C01820=1061.236,135.511,-79.537,172.179,30.450,155.636
C01821=1061.242,135.759,-79.557,172.181,30.453,155.636
C01822=1061.248,136.008,-79.578,172.183,30.455,155.637
C01823=1061.253,136.258,-79.599,172.185,30.458,155.637
C01824=1061.259,136.507,-79.619,172.186,30.461,155.638
C01825=1061.266,136.756,-79.641,172.188,30.463,155.638
C01826=1061.271,137.005,-79.661,172.190,30.466,155.638
C01827=1061.278,137.254,-79.682,172.192,30.469,155.639
C01828=1061.283,137.503,-79.703,172.193,30.471,155.639
C01829=1061.289,137.751,-79.724,172.195,30.474,155.640
C01830=1061.295,138.001,-79.745,172.197,30.477,155.640
C01831=1061.300,138.250,-79.765,172.199,30.480,155.640
C01832=1061.307,138.499,-79.787,172.201,30.482,155.641
C01833=1061.313,138.748,-79.807,172.202,30.485,155.641
C01834=1061.319,138.997,-79.828,172.204,30.488,155.642
C01835=1061.324,139.246,-79.849,172.205,30.490,155.642
C01836=1061.331,139.495,-79.870,172.207,30.493,155.643
C01837=1061.336,139.744,-79.891,172.208,30.495,155.643
C01838=1061.342,139.993,-79.912,172.210,30.498,155.643
C01839=1061.348,140.243,-79.933,172.212,30.501,155.644
C01840=1061.353,140.491,-79.954,172.214,30.503,155.644
C01841=1061.360,140.741,-79.974,172.215,30.507,155.645
C01842=1061.365,140.989,-79.996,172.217,30.509,155.645
C01843=1061.371,141.239,-80.017,172.219,30.512,155.646
C01844=1061.377,141.488,-80.038,172.221,30.515,155.646
C01845=1061.383,141.737,-80.059,172.223,30.517,155.646
C01846=1061.388,141.986,-80.080,172.224,30.520,155.647
C01847=1061.395,142.270,-80.104,172.226,30.523,155.647
C01848=1061.402,142.554,-80.128,172.229,30.526,155.648
C01849=1061.409,142.839,-80.152,172.231,30.529,155.648
C01850=1061.416,143.123,-80.176,172.232,30.533,155.649
C01851=1061.421,143.372,-80.197,172.234,30.535,155.649
C01852=1061.427,143.621,-80.219,172.236,30.538,155.650
C01853=1061.433,143.870,-80.240,172.238,30.541,155.650
C01854=1061.438,144.120,-80.261,172.239,30.543,155.650
C01855=1061.444,144.368,-80.282,172.241,30.546,155.651
C01856=1061.450,144.617,-80.304,172.243,30.549,155.651
C01857=1061.455,144.866,-80.324,172.245,30.551,155.652
C01858=1061.462,145.115,-80.345,172.246,30.554,155.652
C01859=1061.468,145.364,-80.367,172.248,30.557,155.653
C01860=1061.474,145.613,-80.388,172.250,30.560,155.653
C01861=1061.480,145.863,-80.409,172.252,30.563,155.653
C01862=1061.486,146.111,-80.430,172.254,30.565,155.654
C01863=1061.492,146.361,-80.452,172.255,30.568,155.654
C01864=1061.497,146.610,-80.473,172.257,30.571,155.655
C01865=1061.503,146.859,-80.494,172.259,30.573,155.655
C01866=1061.509,147.107,-80.515,172.261,30.576,155.655
C01867=1061.515,147.357,-80.537,172.262,30.579,155.656
C01868=1061.522,147.605,-80.558,172.264,30.581,155.656
C01869=1061.527,147.855,-80.579,172.266,30.584,155.657
C01870=1061.532,148.104,-80.601,172.268,30.587,155.657
C01871=1061.538,148.353,-80.622,172.270,30.590,155.658
C01872=1061.544,148.602,-80.644,172.271,30.592,155.658
C01873=1061.550,148.850,-80.665,172.273,30.595,155.658
C01874=1061.556,149.100,-80.687,172.275,30.598,155.659
C01875=1061.562,149.349,-80.708,172.277,30.600,155.659
C01876=1061.567,149.598,-80.729,172.278,30.603,155.660
C01877=1061.573,149.847,-80.751,172.280,30.606,155.660
C01878=1061.579,150.096,-80.772,172.282,30.609,155.661
C01879=1061.585,150.345,-80.793,172.284,30.612,155.661
C01880=1061.591,150.594,-80.815,172.286,30.614,155.662
C01881=1061.597,150.843,-80.836,172.287,30.617,155.662
C01882=1061.603,151.092,-80.858,172.289,30.620,155.662
C01883=1061.608,151.341,-80.880,172.291,30.622,155.663
C01884=1061.614,151.590,-80.901,172.294,30.625,155.663
C01885=1061.620,151.839,-80.923,172.295,30.628,155.664
C01886=1061.626,152.087,-80.944,172.297,30.631,155.664
C01887=1061.632,152.337,-80.966,172.299,30.634,155.665
C01888=1061.637,152.585,-80.987,172.301,30.636,155.665
C01889=1061.644,152.834,-81.009,172.302,30.639,155.665
C01890=1061.649,153.084,-81.031,172.304,30.642,155.666
C01891=1061.655,153.332,-81.052,172.306,30.645,155.666
C01892=1061.661,153.582,-81.074,172.308,30.648,155.667
C01893=1061.667,153.831,-81.096,172.310,30.650,155.667
C01894=1061.673,154.079,-81.117,172.311,30.653,155.668
C01895=1061.679,154.329,-81.139,172.313,30.656,155.668
C01896=1061.684,154.578,-81.161,172.315,30.658,155.668
C01897=1061.690,154.827,-81.182,172.317,30.661,155.669
C01898=1061.696,155.076,-81.204,172.318,30.664,155.669
C01899=1061.702,155.325,-81.225,172.320,30.667,155.670
C01900=1061.708,155.573,-81.247,172.322,30.669,155.670
C01901=1061.713,155.822,-81.270,172.324,30.672,155.671
C01902=1061.719,156.072,-81.291,172.326,30.675,155.671
C01903=1061.726,156.321,-81.313,172.327,30.678,155.671
C01904=1061.730,156.570,-81.335,172.330,30.681,155.672
C01905=1061.737,156.819,-81.356,172.332,30.684,155.672
C01906=1061.743,157.068,-81.378,172.334,30.686,155.673
C01907=1061.748,157.316,-81.401,172.336,30.689,155.673
C01908=1061.754,157.565,-81.422,172.337,30.692,155.674
C01909=1061.760,157.815,-81.444,172.339,30.695,155.674
C01910=1061.766,158.063,-81.465,172.341,30.697,155.675
C01911=1061.773,158.348,-81.491,172.343,30.701,155.675
C01912=1061.779,158.631,-81.516,172.345,30.704,155.676
C01913=1061.786,158.915,-81.540,172.347,30.707,155.676
C01914=1061.793,159.200,-81.566,172.349,30.710,155.676
C01915=1061.798,159.448,-81.587,172.351,30.713,155.677
C01916=1061.804,159.698,-81.609,172.353,30.716,155.677
C01917=1061.810,159.946,-81.632,172.355,30.719,155.678
C01918=1061.816,160.196,-81.653,172.357,30.721,155.678
C01919=1061.821,160.444,-81.675,172.359,30.724,155.679
C01920=1061.827,160.693,-81.697,172.361,30.727,155.679
C01921=1061.834,160.942,-81.719,172.362,30.729,155.679
C01922=1061.839,161.192,-81.741,172.364,30.732,155.680
C01923=1061.845,161.440,-81.763,172.366,30.735,155.680
C01924=1061.850,161.689,-81.786,172.368,30.738,155.681
C01925=1061.856,161.938,-81.809,172.369,30.741,155.681
C01926=1061.862,162.187,-81.830,172.371,30.744,155.682
C01927=1061.867,162.436,-81.852,172.374,30.747,155.682
C01928=1061.873,162.685,-81.875,172.376,30.750,155.683
C01929=1061.879,162.934,-81.897,172.378,30.752,155.683
C01930=1061.884,163.182,-81.919,172.379,30.756,155.684
C01931=1061.889,163.432,-81.941,172.381,30.758,155.684
C01932=1061.896,163.680,-81.964,172.383,30.761,155.685
C01933=1061.901,163.930,-81.986,172.385,30.764,155.685
C01934=1061.907,164.178,-82.009,172.386,30.767,155.685
C01935=1061.913,164.427,-82.030,172.388,30.770,155.686
C01936=1061.918,164.676,-82.053,172.390,30.773,155.686
C01937=1061.924,164.926,-82.075,172.393,30.775,155.687
C01938=1061.929,165.174,-82.098,172.395,30.779,155.687
C01939=1061.935,165.423,-82.120,172.396,30.781,155.688
C01940=1061.941,165.672,-82.143,172.398,30.785,155.688
C01941=1061.946,165.922,-82.165,172.400,30.787,155.689
C01942=1061.952,166.169,-82.187,172.402,30.790,155.689
C01943=1061.958,166.419,-82.209,172.403,30.793,155.690
C01944=1061.963,166.668,-82.232,172.405,30.796,155.690
C01945=1061.970,166.916,-82.254,172.407,30.798,155.691
C01946=1061.975,167.166,-82.277,172.410,30.802,155.691
C01947=1061.981,167.415,-82.299,172.412,30.804,155.691
C01948=1061.986,167.664,-82.321,172.413,30.808,155.692
C01949=1061.992,167.912,-82.344,172.415,30.810,155.692
C01950=1061.998,168.161,-82.367,172.417,30.813,155.693
C01951=1062.003,168.411,-82.389,172.419,30.816,155.693
C01952=1062.009,168.660,-82.412,172.421,30.819,155.694
C01953=1062.016,168.908,-82.434,172.423,30.822,155.694
C01954=1062.020,169.157,-82.456,172.425,30.825,155.695
C01955=1062.026,169.406,-82.479,172.427,30.827,155.695
C01956=1062.033,169.654,-82.501,172.429,30.830,155.696
C01957=1062.038,169.904,-82.524,172.430,30.833,155.696
C01958=1062.044,170.153,-82.546,172.432,30.836,155.696
C01959=1062.049,170.402,-82.569,172.434,30.839,155.697
C01960=1062.055,170.651,-82.592,172.437,30.842,155.697
C01961=1062.061,170.900,-82.614,172.439,30.845,155.698
C01962=1062.067,171.148,-82.637,172.440,30.848,155.698
C01963=1062.072,171.397,-82.660,172.442,30.850,155.699
C01964=1062.078,171.646,-82.682,172.444,30.853,155.699
C01965=1062.084,171.895,-82.704,172.446,30.856,155.700
C01966=1062.090,172.144,-82.727,172.448,30.859,155.700
C01967=1062.096,172.393,-82.750,172.450,30.862,155.701
C01968=1062.101,172.642,-82.773,172.452,30.865,155.701
C01969=1062.108,172.890,-82.795,172.454,30.868,155.702
C01970=1062.113,173.140,-82.818,172.456,30.871,155.702
C01971=1062.119,173.389,-82.840,172.457,30.874,155.702
C01972=1062.125,173.638,-82.863,172.460,30.876,155.703
C01973=1062.130,173.887,-82.886,172.462,30.880,155.703
C01974=1062.137,174.135,-82.909,172.464,30.882,155.704
C01975=1062.143,174.419,-82.934,172.467,30.886,155.704
C01976=1062.150,174.703,-82.960,172.468,30.889,155.705
C01977=1062.156,174.986,-82.987,172.471,30.892,155.705
C01978=1062.163,175.270,-83.012,172.473,30.895,155.706
C01979=1062.169,175.518,-83.035,172.475,30.898,155.706
C01980=1062.175,175.767,-83.058,172.476,30.901,155.707
C01981=1062.180,176.016,-83.081,172.479,30.904,155.707
C01982=1062.186,176.265,-83.104,172.481,30.907,155.708
C01983=1062.192,176.514,-83.126,172.483,30.910,155.708
C01984=1062.198,176.763,-83.149,172.485,30.912,155.709
C01985=1062.204,177.012,-83.172,172.486,30.915,155.709
C01986=1062.210,177.261,-83.195,172.489,30.919,155.710
C01987=1062.216,177.510,-83.218,172.491,30.921,155.710
C01988=1062.222,177.759,-83.241,172.493,30.924,155.710
C01989=1062.228,178.008,-83.264,172.495,30.927,155.711
C01990=1062.233,178.257,-83.287,172.497,30.930,155.711
C01991=1062.240,178.505,-83.309,172.499,30.932,155.712
C01992=1062.246,178.754,-83.332,172.501,30.936,155.712
C01993=1062.251,179.003,-83.355,172.503,30.938,155.713
C01994=1062.257,179.252,-83.378,172.505,30.941,155.713
C01995=1062.263,179.501,-83.401,172.507,30.944,155.714
C01996=1062.269,179.749,-83.425,172.509,30.947,155.714
C01997=1062.275,179.998,-83.447,172.511,30.950,155.715
C01998=1062.282,180.247,-83.470,172.513,30.953,155.715
C01999=1062.287,180.496,-83.493,172.516,30.956,155.715
C02000=1062.293,180.745,-83.516,172.517,30.959,155.716
C02001=1062.299,180.994,-83.539,172.519,30.961,155.716
C02002=1062.305,181.243,-83.562,172.521,30.964,155.717
C02003=1062.311,181.491,-83.586,172.524,30.967,155.717
C02004=1062.316,181.740,-83.609,172.525,30.970,155.718
C02005=1062.323,181.989,-83.631,172.527,30.973,155.718
C02006=1062.329,182.238,-83.654,172.529,30.976,155.719
C02007=1062.335,182.487,-83.677,172.532,30.979,155.719
C02008=1062.341,182.735,-83.701,172.534,30.981,155.720
C02009=1062.347,182.984,-83.724,172.535,30.984,155.720
C02010=1062.353,183.234,-83.747,172.538,30.987,155.720
C02011=1062.359,183.483,-83.770,172.540,30.990,155.721
C02012=1062.364,183.732,-83.793,172.542,30.993,155.721
C02013=1062.370,183.980,-83.817,172.544,30.996,155.722
C02014=1062.376,184.229,-83.840,172.546,30.999,155.722
C02015=1062.383,184.478,-83.862,172.548,31.002,155.723
C02016=1062.389,184.727,-83.887,172.550,31.005,155.723
C02017=1062.394,184.976,-83.910,172.552,31.008,155.724
C02018=1062.399,185.225,-83.933,172.555,31.011,155.724
C02019=1062.405,185.473,-83.957,172.556,31.014,155.725
C02020=1062.411,185.722,-83.980,172.558,31.017,155.725
C02021=1062.416,185.971,-84.004,172.561,31.020,155.726
C02022=1062.422,186.220,-84.027,172.563,31.023,155.726
C02023=1062.428,186.469,-84.050,172.565,31.026,155.727
C02024=1062.434,186.718,-84.075,172.566,31.029,155.727
C02025=1062.439,186.967,-84.098,172.569,31.032,155.728
C02026=1062.445,187.215,-84.121,172.571,31.035,155.728
C02027=1062.450,187.464,-84.145,172.573,31.038,155.729
C02028=1062.456,187.712,-84.168,172.575,31.041,155.729
C02029=1062.461,187.962,-84.192,172.577,31.044,155.730
C02030=1062.468,188.211,-84.216,172.579,31.048,155.730
C02031=1062.474,188.459,-84.239,172.581,31.050,155.731
C02032=1062.479,188.708,-84.263,172.584,31.053,155.731
C02033=1062.485,188.957,-84.286,172.585,31.057,155.732
C02034=1062.490,189.206,-84.310,172.587,31.059,155.732
C02035=1062.496,189.454,-84.333,172.590,31.063,155.733
C02036=1062.503,189.703,-84.357,172.592,31.066,155.733
C02037=1062.508,189.952,-84.382,172.594,31.068,155.734
C02038=1062.514,190.201,-84.405,172.595,31.072,155.734
C02039=1062.520,190.484,-84.432,172.598,31.075,155.735
C02040=1062.527,190.768,-84.458,172.601,31.079,155.735
C02041=1062.533,191.050,-84.486,172.603,31.082,155.736
C02042=1062.540,191.334,-84.513,172.606,31.086,155.736
C02043=1062.546,191.583,-84.536,172.607,31.089,155.737
C02044=1062.551,191.831,-84.561,172.610,31.091,155.737
C02045=1062.557,192.080,-84.584,172.612,31.095,155.738
C02046=1062.563,192.329,-84.608,172.614,31.098,155.738
C02047=1062.569,192.578,-84.632,172.617,31.101,155.739
C02048=1062.575,192.826,-84.655,172.618,31.104,155.739
C02049=1062.580,193.075,-84.679,172.620,31.107,155.740
C02050=1062.586,193.324,-84.703,172.623,31.110,155.740
C02051=1062.591,193.573,-84.727,172.625,31.113,155.741
C02052=1062.597,193.822,-84.750,172.627,31.116,155.741
C02053=1062.603,194.071,-84.775,172.629,31.120,155.742
C02054=1062.609,194.319,-84.798,172.631,31.122,155.742
C02055=1062.615,194.568,-84.822,172.633,31.125,155.743
C02056=1062.621,194.817,-84.847,172.636,31.129,155.743
C02057=1062.627,195.066,-84.870,172.638,31.131,155.744
C02058=1062.632,195.314,-84.894,172.639,31.135,155.744
C02059=1062.639,195.563,-84.918,172.642,31.138,155.745
C02060=1062.644,195.812,-84.942,172.644,31.140,155.745
C02061=1062.650,196.060,-84.966,172.647,31.144,155.746
C02062=1062.656,196.310,-84.990,172.649,31.147,155.746
C02063=1062.662,196.558,-85.013,172.650,31.150,155.747
C02064=1062.668,196.808,-85.038,172.653,31.153,155.747
C02065=1062.674,197.056,-85.062,172.655,31.156,155.748
C02066=1062.679,197.305,-85.086,172.657,31.159,155.748
C02067=1062.686,197.554,-85.110,172.660,31.162,155.749
C02068=1062.691,197.802,-85.134,172.661,31.165,155.749
C02069=1062.697,198.050,-85.158,172.664,31.169,155.750
C02070=1062.703,198.300,-85.183,172.666,31.171,155.750
C02071=1062.709,198.548,-85.206,172.668,31.174,155.751
C02072=1062.714,198.798,-85.230,172.671,31.178,155.751
C02073=1062.720,199.046,-85.254,172.672,31.180,155.752
C02074=1062.726,199.295,-85.278,172.675,31.184,155.752
C02075=1062.732,199.544,-85.302,172.677,31.187,155.753
C02076=1062.738,199.793,-85.327,172.679,31.190,155.753
C02077=1062.744,200.041,-85.350,172.682,31.193,155.754
C02078=1062.750,200.290,-85.375,172.683,31.196,155.754
C02079=1062.756,200.539,-85.399,172.686,31.199,155.755
C02080=1062.762,200.787,-85.424,172.688,31.202,155.755
C02081=1062.768,201.036,-85.448,172.690,31.205,155.756
C02082=1062.774,201.284,-85.472,172.693,31.209,155.756
C02083=1062.780,201.534,-85.497,172.694,31.211,155.757
C02084=1062.786,201.782,-85.520,172.697,31.214,155.757
C02085=1062.792,202.031,-85.545,172.699,31.218,155.758
C02086=1062.797,202.280,-85.569,172.702,31.221,155.758
C02087=1062.804,202.529,-85.593,172.704,31.224,155.759
C02088=1062.809,202.777,-85.617,172.705,31.227,155.759
C02089=1062.815,203.026,-85.643,172.708,31.230,155.760
C02090=1062.820,203.275,-85.667,172.710,31.233,155.760
C02091=1062.826,203.524,-85.692,172.713,31.237,155.761
C02092=1062.832,203.772,-85.715,172.715,31.240,155.761
C02093=1062.838,204.021,-85.740,172.717,31.243,155.762
C02094=1062.844,204.269,-85.765,172.719,31.246,155.763
C02095=1062.850,204.519,-85.789,172.721,31.250,155.763
C02096=1062.855,204.767,-85.814,172.724,31.253,155.764
C02097=1062.861,205.017,-85.838,172.726,31.256,155.764
C02098=1062.867,205.264,-85.863,172.728,31.259,155.765
C02099=1062.873,205.514,-85.887,172.730,31.262,155.765
C02100=1062.879,205.762,-85.912,172.733,31.265,155.766
C02101=1062.884,206.011,-85.936,172.735,31.268,155.766
C02102=1062.890,206.259,-85.961,172.738,31.272,155.767
C02103=1062.915,207.308,-86.065,172.906,31.353,155.774
C02104=1062.920,207.532,-86.088,172.908,31.357,155.775
C02105=1062.926,207.757,-86.110,172.910,31.361,155.775
C02106=1062.931,207.982,-86.134,172.911,31.364,155.776
C02107=1062.937,208.207,-86.156,172.913,31.368,155.777
C02108=1062.943,208.432,-86.179,172.915,31.372,155.777
C02109=1062.948,208.657,-86.203,172.917,31.376,155.778
C02110=1062.953,208.881,-86.225,172.919,31.379,155.779
C02111=1062.959,209.107,-86.248,172.920,31.383,155.779
C02112=1062.965,209.355,-86.274,172.922,31.387,155.780
C02113=1062.971,209.604,-86.300,172.924,31.391,155.781
C02114=1062.977,209.852,-86.326,172.926,31.395,155.782
C02115=1062.983,210.101,-86.351,172.928,31.399,155.782
C02116=1062.989,210.350,-86.376,172.930,31.404,155.783
C02117=1062.996,210.598,-86.402,172.932,31.407,155.784
C02118=1063.001,210.847,-86.428,172.934,31.412,155.784
C02119=1063.008,211.095,-86.454,172.936,31.415,155.785
C02120=1063.014,211.344,-86.479,172.937,31.420,155.786
C02121=1063.019,211.593,-86.505,172.939,31.423,155.787
C02122=1063.025,211.842,-86.530,172.942,31.428,155.787
C02123=1063.032,212.090,-86.556,172.944,31.432,155.788
C02124=1063.038,212.338,-86.582,172.946,31.436,155.789
C02125=1063.044,212.587,-86.608,172.947,31.440,155.790
C02126=1063.050,212.836,-86.633,172.949,31.444,155.790
C02127=1063.055,213.085,-86.659,172.952,31.448,155.791
C02128=1063.062,213.333,-86.685,172.954,31.452,155.792
C02129=1063.068,213.582,-86.710,172.956,31.456,155.792
C02130=1063.073,213.831,-86.736,172.957,31.460,155.793
C02131=1063.080,214.079,-86.762,172.959,31.464,155.794
C02132=1063.085,214.328,-86.788,172.962,31.469,155.795
C02133=1063.092,214.576,-86.814,172.964,31.472,155.795
C02134=1063.097,214.825,-86.840,172.966,31.477,155.796
C02135=1063.104,215.073,-86.866,172.967,31.480,155.797
C02136=1063.109,215.322,-86.892,172.969,31.485,155.798
C02137=1063.116,215.570,-86.918,172.972,31.488,155.798
C02138=1063.122,215.819,-86.943,172.974,31.493,155.799
C02139=1063.128,216.068,-86.969,172.976,31.496,155.800
C02140=1063.134,216.316,-86.995,172.977,31.501,155.801
C02141=1063.140,216.565,-87.021,172.979,31.504,155.801
C02142=1063.146,216.813,-87.047,172.982,31.509,155.802
C02143=1063.152,217.062,-87.073,172.984,31.513,155.803
C02144=1063.158,217.310,-87.099,172.986,31.517,155.803
C02145=1063.164,217.559,-87.125,172.987,31.521,155.804
C02146=1063.170,217.808,-87.151,172.990,31.525,155.805
C02147=1063.176,218.056,-87.178,172.992,31.529,155.806
C02148=1063.182,218.305,-87.203,172.994,31.533,155.806
C02149=1063.188,218.553,-87.230,172.996,31.537,155.807
C02150=1063.194,218.802,-87.255,172.998,31.541,155.808
C02151=1063.200,219.050,-87.282,173.000,31.545,155.808
C02152=1063.206,219.299,-87.307,173.002,31.549,155.809
C02153=1063.212,219.547,-87.334,173.004,31.553,155.810
C02154=1063.219,219.797,-87.359,173.007,31.557,155.811
C02155=1063.225,220.045,-87.386,173.008,31.561,155.811
C02156=1063.231,220.293,-87.412,173.010,31.565,155.812
C02157=1063.237,220.542,-87.438,173.012,31.569,155.813
C02158=1063.243,220.790,-87.464,173.015,31.573,155.813
C02159=1063.249,221.039,-87.491,173.017,31.577,155.814
C02160=1063.254,221.266,-87.515,173.019,31.581,155.815
C02161=1063.260,221.494,-87.539,173.020,31.584,155.815
C02162=1063.265,221.721,-87.562,173.022,31.588,155.816
C02163=1063.271,221.948,-87.587,173.024,31.591,155.817
C02164=1063.277,222.176,-87.611,173.026,31.595,155.817
C02165=1063.282,222.403,-87.635,173.028,31.599,155.818
C02166=1063.288,222.630,-87.659,173.030,31.602,155.819
C02167=1063.293,222.858,-87.683,173.031,31.606,155.820
C02168=1063.299,223.106,-87.710,173.034,31.611,155.820
C02169=1063.305,223.355,-87.736,173.036,31.614,155.821
C02170=1063.310,223.603,-87.763,173.038,31.619,155.822
C02171=1063.318,223.852,-87.789,173.041,31.622,155.822
C02172=1063.323,224.100,-87.816,173.042,31.627,155.823
C02173=1063.329,224.349,-87.842,173.044,31.630,155.824
C02174=1063.335,224.598,-87.868,173.046,31.635,155.825
C02175=1063.341,224.846,-87.894,173.049,31.638,155.825
C02176=1063.347,225.095,-87.921,173.051,31.642,155.826
C02177=1063.353,225.343,-87.948,173.053,31.646,155.827
C02178=1063.359,225.592,-87.975,173.055,31.650,155.827
C02179=1063.365,225.840,-88.001,173.057,31.655,155.828
C02180=1063.372,226.089,-88.028,173.059,31.658,155.829
C02181=1063.378,226.337,-88.054,173.061,31.662,155.830
C02182=1063.383,226.585,-88.081,173.064,31.666,155.830
C02183=1063.389,226.834,-88.108,173.066,31.670,155.831
C02184=1063.395,227.084,-88.134,173.067,31.674,155.832
C02185=1063.402,227.332,-88.160,173.070,31.678,155.832
C02186=1063.408,227.580,-88.187,173.072,31.682,155.833
C02187=1063.414,227.829,-88.214,173.074,31.686,155.834
C02188=1063.420,228.077,-88.240,173.077,31.690,155.835
C02189=1063.425,228.326,-88.267,173.078,31.694,155.835
C02190=1063.433,228.574,-88.293,173.080,31.698,155.836
C02191=1063.439,228.822,-88.321,173.083,31.702,155.837
C02192=1063.444,229.071,-88.347,173.085,31.706,155.838
C02193=1063.451,229.320,-88.374,173.087,31.710,155.838
C02194=1063.457,229.568,-88.401,173.090,31.714,155.839
C02195=1063.462,229.816,-88.428,173.091,31.718,155.840
C02196=1063.469,230.065,-88.455,173.093,31.721,155.840
C02197=1063.475,230.314,-88.481,173.096,31.726,155.841
C02198=1063.480,230.562,-88.508,173.098,31.730,155.842
C02199=1063.487,230.811,-88.535,173.100,31.734,155.843
C02200=1063.492,231.060,-88.562,173.103,31.738,155.843
C02201=1063.499,231.307,-88.589,173.104,31.742,155.844
C02202=1063.505,231.556,-88.616,173.106,31.746,155.845
C02203=1063.511,231.805,-88.643,173.109,31.749,155.845
C02204=1063.516,232.053,-88.669,173.111,31.754,155.846
C02205=1063.523,232.302,-88.696,173.113,31.757,155.847
C02206=1063.529,232.550,-88.724,173.116,31.762,155.848
C02207=1063.535,232.798,-88.750,173.117,31.765,155.848
C02208=1063.541,233.047,-88.777,173.119,31.770,155.849
C02209=1063.547,233.296,-88.804,173.122,31.774,155.850
C02210=1063.553,233.544,-88.832,173.124,31.777,155.850
C02211=1063.559,233.792,-88.858,173.127,31.782,155.851
C02212=1063.564,234.041,-88.886,173.129,31.785,155.852
C02213=1063.571,234.290,-88.913,173.131,31.790,155.853
C02214=1063.577,234.538,-88.940,173.133,31.793,155.853
C02215=1063.583,234.786,-88.967,173.135,31.798,155.854
C02216=1063.588,235.010,-88.991,173.137,31.801,155.855
C02217=1063.594,235.233,-89.016,173.139,31.804,155.855
C02218=1063.599,235.457,-89.040,173.141,31.808,155.856
C02219=1063.605,235.680,-89.064,173.144,31.812,155.857
C02220=1063.610,235.903,-89.089,173.146,31.815,155.857
C02221=1063.616,236.127,-89.113,173.147,31.819,155.858
C02222=1063.621,236.350,-89.138,173.149,31.822,155.859
C02223=1063.626,236.574,-89.163,173.151,31.826,155.859
C02224=1063.632,236.821,-89.190,173.154,31.830,155.860
C02225=1063.638,237.070,-89.217,173.156,31.834,155.861
C02226=1063.644,237.318,-89.244,173.158,31.838,155.861
C02227=1063.651,237.567,-89.271,173.160,31.842,155.862
C02228=1063.657,237.815,-89.299,173.162,31.846,155.863
C02229=1063.662,238.064,-89.326,173.165,31.850,155.864
C02230=1063.669,238.312,-89.354,173.167,31.853,155.864
C02231=1063.675,238.561,-89.381,173.169,31.858,155.865
C02232=1063.681,238.809,-89.408,173.172,31.861,155.866
C02233=1063.687,239.058,-89.437,173.174,31.865,155.866
C02234=1063.693,239.306,-89.463,173.176,31.869,155.867
C02235=1063.699,239.554,-89.491,173.178,31.873,155.868
C02236=1063.705,239.803,-89.518,173.180,31.877,155.868
C02237=1063.711,240.052,-89.546,173.183,31.881,155.869
C02238=1063.717,240.299,-89.573,173.185,31.885,155.870
C02239=1063.724,240.548,-89.600,173.188,31.889,155.871
C02240=1063.729,240.796,-89.628,173.190,31.893,155.871
C02241=1063.736,241.045,-89.656,173.192,31.897,155.872
C02242=1063.742,241.294,-89.683,173.194,31.900,155.873
C02243=1063.748,241.542,-89.710,173.197,31.905,155.874
C02244=1063.754,241.790,-89.739,173.199,31.908,155.874
C02245=1063.760,242.039,-89.765,173.201,31.912,155.875
C02246=1063.766,242.287,-89.793,173.204,31.917,155.876
C02247=1063.772,242.535,-89.821,173.206,31.920,155.876
C02248=1063.778,242.784,-89.849,173.208,31.925,155.877
C02249=1063.784,243.033,-89.876,173.210,31.928,155.878
C02250=1063.790,243.281,-89.904,173.213,31.932,155.878
C02251=1063.796,243.530,-89.932,173.215,31.936,155.879
C02252=1063.802,243.777,-89.959,173.218,31.940,155.880
C02253=1063.808,244.026,-89.988,173.220,31.944,155.881
C02254=1063.814,244.274,-90.014,173.222,31.948,155.881
C02255=1063.820,244.523,-90.043,173.224,31.952,155.882
C02256=1063.827,244.772,-90.070,173.226,31.956,155.883
C02257=1063.832,245.020,-90.098,173.229,31.960,155.884
C02258=1063.839,245.268,-90.126,173.231,31.964,155.884
C02259=1063.844,245.516,-90.154,173.234,31.968,155.885
C02260=1063.851,245.765,-90.182,173.236,31.972,155.886
C02261=1063.857,246.013,-90.210,173.239,31.976,155.886
C02262=1063.862,246.261,-90.238,173.241,31.980,155.887
C02263=1063.869,246.510,-90.266,173.243,31.984,155.888
C02264=1063.874,246.758,-90.294,173.245,31.988,155.889
C02265=1063.880,247.007,-90.322,173.248,31.992,155.889
C02266=1063.886,247.255,-90.350,173.250,31.996,155.890
C02267=1063.892,247.503,-90.378,173.253,32.000,155.891
C02268=1063.898,247.752,-90.406,173.255,32.004,155.892
C02269=1063.904,248.000,-90.433,173.257,32.007,155.892
C02270=1063.910,248.248,-90.462,173.259,32.012,155.893
C02271=1063.916,248.497,-90.490,173.261,32.015,155.894
C02272=1063.921,248.717,-90.515,173.264,32.019,155.894
C02273=1063.926,248.937,-90.540,173.266,32.023,155.895
C02274=1063.932,249.157,-90.565,173.268,32.026,155.896
C02275=1063.937,249.378,-90.590,173.270,32.030,155.896
C02276=1063.942,249.598,-90.614,173.272,32.033,155.897
C02277=1063.947,249.818,-90.640,173.275,32.037,155.898
C02278=1063.953,250.038,-90.664,173.277,32.040,155.898
C02279=1063.957,250.259,-90.689,173.278,32.044,155.899
C02280=1063.964,250.507,-90.718,173.281,32.048,155.900
C02281=1063.970,250.755,-90.746,173.283,32.052,155.900
C02282=1063.976,251.003,-90.774,173.286,32.056,155.901
C02283=1063.982,251.252,-90.802,173.288,32.060,155.902
C02284=1063.988,251.500,-90.832,173.291,32.064,155.902
C02285=1063.993,251.748,-90.859,173.293,32.068,155.903
C02286=1064.000,251.997,-90.887,173.296,32.072,155.904
C02287=1064.006,252.246,-90.916,173.297,32.076,155.905
C02288=1064.012,252.493,-90.944,173.300,32.080,155.905
C02289=1064.017,252.742,-90.973,173.302,32.083,155.906
C02290=1064.023,252.991,-91.001,173.305,32.088,155.907
C02291=1064.030,253.238,-91.029,173.307,32.091,155.908
C02292=1064.036,253.487,-91.058,173.310,32.096,155.908
C02293=1064.042,253.735,-91.086,173.312,32.099,155.909
C02294=1064.048,253.983,-91.115,173.315,32.103,155.910
C02295=1064.054,254.232,-91.143,173.317,32.107,155.911
C02296=1064.060,254.481,-91.171,173.319,32.111,155.911
C02297=1064.066,254.728,-91.199,173.322,32.115,155.912
C02298=1064.072,254.977,-91.228,173.324,32.119,155.913
C02299=1064.078,255.225,-91.257,173.327,32.123,155.913
C02300=1064.084,255.474,-91.285,173.329,32.127,155.914
C02301=1064.091,255.722,-91.314,173.332,32.131,155.915
C02302=1064.097,255.970,-91.342,173.335,32.135,155.915
C02303=1064.102,256.218,-91.371,173.337,32.139,155.916
C02304=1064.109,256.466,-91.399,173.339,32.143,155.917
C02305=1064.115,256.714,-91.428,173.341,32.146,155.918
C02306=1064.121,256.963,-91.456,173.344,32.151,155.918
C02307=1064.127,257.211,-91.485,173.346,32.154,155.919
C02308=1064.133,257.460,-91.514,173.349,32.158,155.920
C02309=1064.140,257.708,-91.543,173.352,32.162,155.921
C02310=1064.145,257.957,-91.571,173.354,32.166,155.921
C02311=1064.151,258.204,-91.600,173.357,32.170,155.922
C02312=1064.158,258.453,-91.627,173.359,32.174,155.923
C02313=1064.164,258.701,-91.656,173.361,32.178,155.923
C02314=1064.170,258.949,-91.685,173.364,32.181,155.924
C02315=1064.176,259.198,-91.714,173.366,32.186,155.925
C02316=1064.182,259.446,-91.743,173.369,32.189,155.926
C02317=1064.189,259.694,-91.772,173.371,32.193,155.926
C02318=1064.195,259.943,-91.800,173.374,32.197,155.927
C02319=1064.201,260.191,-91.829,173.377,32.201,155.928
C02320=1064.207,260.439,-91.858,173.379,32.205,155.928
C02321=1064.213,260.688,-91.887,173.382,32.209,155.929
C02322=1064.220,260.936,-91.915,173.384,32.213,155.930
C02323=1064.226,261.184,-91.944,173.386,32.217,155.931
C02324=1064.233,261.432,-91.973,173.389,32.220,155.931
C02325=1064.239,261.681,-92.001,173.391,32.225,155.932
C02326=1064.245,261.929,-92.030,173.394,32.228,155.933
C02327=1064.251,262.177,-92.059,173.397,32.232,155.933
C02328=1064.257,262.397,-92.085,173.399,32.236,155.934
C02329=1064.262,262.615,-92.111,173.401,32.239,155.935
C02330=1064.267,262.835,-92.136,173.404,32.243,155.935
C02331=1064.273,263.053,-92.161,173.406,32.246,155.936
C02332=1064.278,263.273,-92.187,173.408,32.249,155.937
C02333=1064.284,263.492,-92.213,173.410,32.252,155.937
C02334=1064.289,263.711,-92.238,173.412,32.256,155.938
C02335=1064.295,263.930,-92.264,173.414,32.260,155.938
C02336=1064.301,264.178,-92.293,173.417,32.263,155.939
C02337=1064.307,264.426,-92.322,173.420,32.268,155.940
C02338=1064.313,264.675,-92.352,173.422,32.271,155.941
C02339=1064.319,264.923,-92.381,173.425,32.276,155.941
C02340=1064.325,265.171,-92.410,173.428,32.280,155.942
C02341=1064.332,265.419,-92.439,173.430,32.283,155.943
C02342=1064.337,265.668,-92.469,173.433,32.287,155.944
C02343=1064.343,265.916,-92.498,173.436,32.291,155.944
C02344=1064.350,266.164,-92.527,173.437,32.295,155.945
C02345=1064.356,266.412,-92.556,173.440,32.299,155.946
C02346=1064.361,266.660,-92.586,173.443,32.303,155.946
C02347=1064.368,266.908,-92.615,173.445,32.307,155.947
C02348=1064.374,267.157,-92.644,173.448,32.311,155.948
C02349=1064.379,267.405,-92.673,173.451,32.315,155.949
C02350=1064.386,267.653,-92.702,173.453,32.319,155.949
C02351=1064.392,267.901,-92.731,173.456,32.323,155.950
C02352=1064.398,268.149,-92.762,173.459,32.327,155.951
C02353=1064.404,268.397,-92.791,173.461,32.331,155.952
C02354=1064.410,268.645,-92.820,173.464,32.335,155.952
C02355=1064.417,268.894,-92.849,173.466,32.339,155.953
C02356=1064.422,269.143,-92.879,173.468,32.343,155.954
C02357=1064.429,269.391,-92.908,173.471,32.347,155.954
C02358=1064.435,269.639,-92.938,173.474,32.351,155.955
C02359=1064.441,269.887,-92.967,173.476,32.354,155.956
C02360=1064.446,270.135,-92.997,173.479,32.359,155.957
C02361=1064.453,270.383,-93.027,173.482,32.363,155.957
C02362=1064.459,270.631,-93.056,173.485,32.367,155.958
C02363=1064.465,270.879,-93.085,173.487,32.370,155.959
C02364=1064.472,271.128,-93.115,173.490,32.375,155.960
C02365=1064.477,271.376,-93.145,173.493,32.378,155.960
C02366=1064.484,271.624,-93.174,173.495,32.382,155.961
C02367=1064.489,271.872,-93.204,173.497,32.386,155.962
C02368=1064.496,272.120,-93.233,173.500,32.390,155.963
C02369=1064.501,272.368,-93.263,173.503,32.394,155.963
C02370=1064.508,272.617,-93.293,173.505,32.398,155.964
C02371=1064.514,272.865,-93.323,173.508,32.402,155.965
C02372=1064.520,273.113,-93.353,173.511,32.406,155.965
C02373=1064.526,273.361,-93.382,173.513,32.410,155.966
C02374=1064.532,273.609,-93.412,173.516,32.414,155.967
C02375=1064.538,273.857,-93.442,173.519,32.418,155.968
C02376=1064.545,274.105,-93.472,173.522,32.422,155.968
C02377=1064.551,274.354,-93.501,173.524,32.426,155.969
C02378=1064.556,274.602,-93.532,173.527,32.430,155.970
C02379=1064.563,274.850,-93.561,173.530,32.434,155.971
C02380=1064.568,275.097,-93.591,173.532,32.438,155.971
C02381=1064.575,275.347,-93.621,173.534,32.442,155.972
C02382=1064.581,275.594,-93.651,173.537,32.446,155.973
C02383=1064.587,275.842,-93.681,173.540,32.450,155.974
C02384=1064.593,276.063,-93.707,173.542,32.454,155.974
C02385=1064.598,276.284,-93.734,173.545,32.458,155.975
C02386=1064.603,276.505,-93.761,173.547,32.461,155.976
C02387=1064.609,276.726,-93.787,173.550,32.464,155.976
C02388=1064.614,276.947,-93.814,173.552,32.468,155.977
C02389=1064.620,277.168,-93.842,173.555,32.472,155.978
C02390=1064.625,277.388,-93.868,173.557,32.475,155.978
C02391=1064.630,277.609,-93.895,173.560,32.479,155.979
C02392=1064.637,277.858,-93.925,173.562,32.483,155.980
C02393=1064.643,278.106,-93.954,173.565,32.487,155.981
C02394=1064.649,278.354,-93.985,173.568,32.491,155.981
C02395=1064.655,278.602,-94.015,173.570,32.495,155.982
C02396=1064.662,278.850,-94.045,173.572,32.499,155.983
C02397=1064.667,279.098,-94.075,173.575,32.503,155.983
C02398=1064.674,279.347,-94.106,173.578,32.507,155.984
C02399=1064.679,279.595,-94.136,173.581,32.511,155.985
C02400=1064.686,279.842,-94.166,173.584,32.515,155.986
C02401=1064.692,280.091,-94.196,173.586,32.519,155.986
C02402=1064.698,280.338,-94.227,173.589,32.523,155.987
C02403=1064.704,280.586,-94.257,173.592,32.527,155.988
C02404=1064.710,280.835,-94.287,173.595,32.531,155.989
C02405=1064.716,281.083,-94.317,173.598,32.535,155.989
C02406=1064.722,281.331,-94.348,173.600,32.539,155.990
C02407=1064.728,281.580,-94.379,173.603,32.543,155.991
C02408=1064.735,281.827,-94.408,173.606,32.547,155.992
C02409=1064.741,282.075,-94.439,173.609,32.551,155.993
C02410=1064.747,282.323,-94.469,173.612,32.556,155.993
C02411=1064.753,282.571,-94.500,173.615,32.559,155.994
C02412=1064.759,282.819,-94.530,173.616,32.563,155.995
C02413=1064.765,283.068,-94.561,173.619,32.568,155.996
C02414=1064.771,283.315,-94.591,173.622,32.571,155.996
C02415=1064.777,283.563,-94.622,173.625,32.576,155.997
C02416=1064.783,283.811,-94.653,173.628,32.579,155.998
C02417=1064.789,284.059,-94.683,173.631,32.584,155.999
C02418=1064.796,284.307,-94.714,173.633,32.588,155.999
C02419=1064.801,284.555,-94.744,173.636,32.592,156.000
C02420=1064.807,284.803,-94.775,173.639,32.596,156.001
C02421=1064.814,285.052,-94.805,173.642,32.600,156.002
C02422=1064.819,285.299,-94.836,173.645,32.604,156.002
C02423=1064.826,285.547,-94.867,173.648,32.608,156.003
C02424=1064.832,285.795,-94.898,173.650,32.612,156.004
C02425=1064.838,286.044,-94.928,173.653,32.616,156.005
C02426=1064.844,286.292,-94.959,173.656,32.620,156.005
C02427=1064.851,286.539,-94.990,173.659,32.624,156.006
C02428=1064.857,286.787,-95.020,173.662,32.628,156.007
C02429=1064.863,287.036,-95.051,173.665,32.632,156.008
C02430=1064.869,287.284,-95.081,173.668,32.636,156.008
C02431=1064.876,287.531,-95.113,173.670,32.640,156.009
C02432=1064.882,287.779,-95.143,173.672,32.645,156.010
C02433=1064.888,288.028,-95.174,173.675,32.648,156.011
C02434=1064.894,288.275,-95.205,173.678,32.653,156.012
C02435=1064.901,288.524,-95.236,173.681,32.657,156.012
C02436=1064.906,288.771,-95.266,173.684,32.661,156.013
C02437=1064.913,289.019,-95.298,173.687,32.665,156.014
C02438=1064.918,289.267,-95.328,173.690,32.669,156.015
C02439=1064.925,289.515,-95.360,173.693,32.673,156.015
C02440=1064.931,289.742,-95.388,173.695,32.677,156.016
C02441=1064.936,289.967,-95.416,173.698,32.681,156.017
C02442=1064.942,290.194,-95.444,173.701,32.684,156.018
C02443=1064.948,290.420,-95.473,173.703,32.688,156.018
C02444=1064.953,290.646,-95.501,173.706,32.692,156.019
C02445=1064.959,290.872,-95.529,173.709,32.696,156.020
C02446=1064.965,291.099,-95.557,173.711,32.699,156.020
C02447=1064.970,291.325,-95.586,173.714,32.703,156.021
C02448=1064.976,291.572,-95.617,173.717,32.707,156.022
C02449=1064.982,291.821,-95.648,173.720,32.711,156.023
C02450=1064.988,292.068,-95.679,173.723,32.715,156.023
C02451=1064.994,292.316,-95.711,173.726,32.720,156.024
C02452=1065.001,292.565,-95.742,173.729,32.724,156.025
C02453=1065.007,292.812,-95.773,173.731,32.728,156.026
C02454=1065.013,293.061,-95.804,173.734,32.732,156.027
C02455=1065.019,293.308,-95.835,173.737,32.736,156.027
C02456=1065.025,293.556,-95.867,173.740,32.740,156.028
C02457=1065.032,293.804,-95.898,173.743,32.744,156.029
C02458=1065.037,294.052,-95.929,173.745,32.749,156.030
C02459=1065.044,294.300,-95.960,173.748,32.752,156.030
C02460=1065.051,294.548,-95.992,173.751,32.757,156.031
C02461=1065.056,294.796,-96.023,173.754,32.761,156.032
C02462=1065.062,295.044,-96.054,173.757,32.765,156.033
C02463=1065.068,295.292,-96.086,173.760,32.769,156.034
C02464=1065.075,295.539,-96.117,173.763,32.773,156.034
C02465=1065.081,295.787,-96.149,173.766,32.777,156.035
C02466=1065.087,296.035,-96.181,173.769,32.782,156.036
C02467=1065.093,296.283,-96.211,173.772,32.786,156.037
C02468=1065.099,296.531,-96.243,173.775,32.790,156.038
C02469=1065.106,296.779,-96.275,173.778,32.794,156.038
C02470=1065.111,297.027,-96.306,173.781,32.799,156.039
C02471=1065.118,297.275,-96.338,173.784,32.803,156.040
C02472=1065.124,297.523,-96.370,173.787,32.807,156.041
C02473=1065.130,297.770,-96.401,173.790,32.811,156.042
C02474=1065.136,298.018,-96.433,173.793,32.815,156.042
C02475=1065.142,298.267,-96.465,173.796,32.820,156.043
C02476=1065.147,298.514,-96.497,173.799,32.824,156.044
C02477=1065.154,298.762,-96.528,173.802,32.828,156.045
C02478=1065.160,299.010,-96.560,173.805,32.832,156.046
C02479=1065.165,299.258,-96.592,173.808,32.837,156.046
C02480=1065.172,299.506,-96.623,173.811,32.841,156.047
C02481=1065.178,299.754,-96.655,173.814,32.845,156.048
C02482=1065.184,300.001,-96.688,173.817,32.849,156.049
C02483=1065.190,300.249,-96.720,173.820,32.854,156.050
C02484=1065.197,300.497,-96.751,173.823,32.858,156.051
C02485=1065.203,300.745,-96.783,173.826,32.862,156.051
C02486=1065.208,300.993,-96.815,173.829,32.866,156.052
C02487=1065.214,301.241,-96.847,173.832,32.871,156.053
C02488=1065.221,301.488,-96.879,173.835,32.875,156.054
C02489=1065.227,301.736,-96.911,173.838,32.880,156.055
C02490=1065.233,301.985,-96.943,173.841,32.884,156.056
C02491=1065.238,302.232,-96.975,173.844,32.888,156.056
C02492=1065.245,302.479,-97.007,173.847,32.892,156.057
C02493=1065.251,302.728,-97.039,173.850,32.896,156.058
C02494=1065.257,302.976,-97.071,173.853,32.901,156.059
C02495=1065.264,303.223,-97.104,173.856,32.905,156.060
C02496=1065.269,303.457,-97.133,173.859,32.909,156.060
C02497=1065.275,303.690,-97.163,173.862,32.913,156.061
C02498=1065.281,303.924,-97.193,173.865,32.917,156.062
C02499=1065.286,304.158,-97.224,173.867,32.921,156.063
C02500=1065.293,304.391,-97.254,173.870,32.925,156.064
C02501=1065.298,304.625,-97.285,173.873,32.929,156.064
C02502=1065.304,304.859,-97.315,173.876,32.933,156.065
C02503=1065.310,305.093,-97.345,173.879,32.937,156.066
C02504=1065.316,305.341,-97.378,173.882,32.942,156.067
C02505=1065.323,305.588,-97.409,173.885,32.946,156.068
C02506=1065.329,305.836,-97.442,173.888,32.950,156.068
C02507=1065.335,306.084,-97.474,173.891,32.954,156.069
C02508=1065.341,306.332,-97.507,173.894,32.959,156.070
C02509=1065.347,306.580,-97.539,173.897,32.963,156.071
C02510=1065.354,306.827,-97.571,173.901,32.968,156.072
C02511=1065.360,307.076,-97.603,173.904,32.972,156.073
C02512=1065.366,307.322,-97.636,173.907,32.976,156.073
C02513=1065.372,307.571,-97.668,173.910,32.980,156.074
C02514=1065.378,307.818,-97.700,173.913,32.985,156.075
C02515=1065.385,308.066,-97.733,173.916,32.989,156.076
C02516=1065.391,308.314,-97.765,173.919,32.993,156.077
C02517=1065.398,308.561,-97.797,173.922,32.998,156.078
C02518=1065.404,308.809,-97.830,173.925,33.002,156.078
C02519=1065.411,309.058,-97.862,173.929,33.006,156.079
C02520=1065.417,309.305,-97.895,173.932,33.010,156.080
C02521=1065.423,309.553,-97.928,173.935,33.015,156.081
C02522=1065.429,309.801,-97.960,173.938,33.019,156.082
C02523=1065.435,310.049,-97.993,173.941,33.024,156.083
C02524=1065.442,310.296,-98.025,173.944,33.028,156.083
C02525=1065.449,310.544,-98.057,173.947,33.032,156.084
C02526=1065.455,310.791,-98.090,173.951,33.036,156.085
C02527=1065.461,311.039,-98.122,173.954,33.041,156.086
C02528=1065.467,311.287,-98.155,173.957,33.045,156.087
C02529=1065.474,311.535,-98.188,173.960,33.049,156.088
C02530=1065.480,311.782,-98.220,173.963,33.054,156.088
C02531=1065.487,312.031,-98.254,173.966,33.058,156.089
C02532=1065.493,312.278,-98.286,173.970,33.062,156.090
C02533=1065.499,312.526,-98.318,173.973,33.067,156.091
C02534=1065.505,312.774,-98.351,173.976,33.071,156.092
C02535=1065.512,313.022,-98.384,173.979,33.075,156.093
C02536=1065.519,313.269,-98.416,173.982,33.080,156.093
C02537=1065.526,313.517,-98.449,173.985,33.084,156.094
C02538=1065.532,313.765,-98.482,173.989,33.089,156.095
C02539=1065.538,314.012,-98.515,173.992,33.093,156.096
C02540=1065.544,314.260,-98.548,173.995,33.098,156.097
C02541=1065.550,314.508,-98.581,173.998,33.102,156.098
C02542=1065.556,314.755,-98.613,174.001,33.106,156.099
C02543=1065.562,315.003,-98.647,174.004,33.111,156.099
C02544=1065.568,315.250,-98.680,174.008,33.116,156.100
C02545=1065.575,315.499,-98.714,174.011,33.120,156.101
C02546=1065.581,315.746,-98.747,174.014,33.124,156.102
C02547=1065.586,315.994,-98.780,174.017,33.129,156.103
C02548=1065.593,316.242,-98.813,174.020,33.133,156.104
C02549=1065.599,316.489,-98.846,174.023,33.138,156.105
C02550=1065.605,316.737,-98.880,174.027,33.142,156.106
C02551=1065.612,316.985,-98.913,174.031,33.147,156.107
C02552=1065.618,317.224,-98.945,174.034,33.151,156.107
C02553=1065.623,317.463,-98.978,174.037,33.156,156.108
C02554=1065.629,317.702,-99.009,174.040,33.160,156.109
C02555=1065.635,317.942,-99.041,174.043,33.164,156.110
C02556=1065.641,318.180,-99.073,174.046,33.169,156.111
C02557=1065.648,318.419,-99.105,174.049,33.173,156.112
C02558=1065.653,318.658,-99.138,174.053,33.178,156.113
C02559=1065.659,318.897,-99.170,174.056,33.182,156.114
C02560=1065.665,319.141,-99.203,174.059,33.187,156.114
C02561=1065.672,319.386,-99.236,174.062,33.191,156.115
C02562=1065.677,319.630,-99.268,174.065,33.195,156.116
C02563=1065.683,319.874,-99.302,174.068,33.200,156.117
C02564=1065.689,320.118,-99.335,174.072,33.205,156.118
C02565=1065.696,320.363,-99.368,174.075,33.209,156.119
C02566=1065.702,320.607,-99.401,174.078,33.214,156.120
C02567=1065.708,320.850,-99.434,174.081,33.218,156.121
C02568=1065.714,321.098,-99.467,174.084,33.223,156.122
C02569=1065.721,321.346,-99.501,174.088,33.228,156.123
C02570=1065.727,321.593,-99.535,174.091,33.232,156.123
C02571=1065.733,321.841,-99.568,174.094,33.237,156.124
C02572=1065.740,322.089,-99.602,174.097,33.241,156.125
C02573=1065.746,322.336,-99.635,174.101,33.246,156.126
C02574=1065.752,322.584,-99.669,174.105,33.250,156.127
C02575=1065.759,322.832,-99.702,174.108,33.255,156.128
C02576=1065.765,323.079,-99.736,174.111,33.260,156.129
C02577=1065.772,323.327,-99.770,174.115,33.264,156.130
C02578=1065.777,323.575,-99.803,174.118,33.269,156.131
C02579=1065.785,323.823,-99.837,174.121,33.273,156.132
C02580=1065.790,324.070,-99.871,174.125,33.278,156.133
C02581=1065.797,324.318,-99.905,174.128,33.282,156.133
C02582=1065.803,324.565,-99.938,174.131,33.287,156.134
C02583=1065.809,324.813,-99.972,174.135,33.292,156.135
C02584=1065.816,325.060,-100.006,174.138,33.297,156.136
C02585=1065.822,325.308,-100.040,174.141,33.301,156.137
C02586=1065.829,325.556,-100.073,174.144,33.306,156.138
C02587=1065.835,325.803,-100.107,174.148,33.310,156.139
C02588=1065.841,326.051,-100.142,174.151,33.315,156.140
C02589=1065.848,326.299,-100.176,174.154,33.320,156.141
C02590=1065.854,326.546,-100.210,174.158,33.325,156.142
C02591=1065.862,326.794,-100.243,174.162,33.329,156.143
C02592=1065.867,327.041,-100.277,174.165,33.333,156.144
C02593=1065.874,327.289,-100.312,174.169,33.338,156.144
C02594=1065.880,327.537,-100.345,174.172,33.343,156.145
C02595=1065.887,327.785,-100.379,174.176,33.348,156.146
C02596=1065.893,328.033,-100.413,174.179,33.352,156.147
C02597=1065.900,328.280,-100.447,174.182,33.357,156.148
C02598=1065.906,328.528,-100.481,174.186,33.362,156.149
C02599=1065.913,328.775,-100.515,174.189,33.367,156.150
C02600=1065.919,329.023,-100.549,174.192,33.371,156.151
C02601=1065.926,329.271,-100.584,174.196,33.376,156.152
C02602=1065.933,329.517,-100.618,174.199,33.380,156.153
C02603=1065.939,329.765,-100.652,174.203,33.385,156.154
C02604=1065.945,330.013,-100.687,174.207,33.390,156.155
C02605=1065.952,330.260,-100.720,174.210,33.395,156.156
C02606=1065.959,330.508,-100.755,174.214,33.399,156.157
C02607=1065.965,330.756,-100.789,174.217,33.404,156.158
C02608=1065.971,330.988,-100.821,174.220,33.409,156.159
C02609=1065.977,331.221,-100.853,174.223,33.413,156.159
C02610=1065.984,331.454,-100.885,174.227,33.418,156.160
C02611=1065.989,331.686,-100.918,174.230,33.422,156.161
C02612=1065.995,331.919,-100.950,174.233,33.426,156.162
C02613=1066.001,332.151,-100.983,174.236,33.431,156.163
C02614=1066.007,332.384,-101.016,174.239,33.436,156.164
C02615=1066.013,332.616,-101.048,174.243,33.441,156.165
C02616=1066.019,332.863,-101.082,174.247,33.445,156.166
C02617=1066.026,333.111,-101.117,174.250,33.450,156.167
C02618=1066.032,333.359,-101.152,174.254,33.455,156.168
C02619=1066.038,333.606,-101.186,174.257,33.460,156.169
C02620=1066.045,333.853,-101.221,174.261,33.465,156.170
C02621=1066.051,334.101,-101.255,174.264,33.470,156.171
C02622=1066.058,334.348,-101.290,174.268,33.475,156.172
C02623=1066.064,334.596,-101.325,174.271,33.480,156.173
C02624=1066.070,334.844,-101.359,174.274,33.484,156.174
C02625=1066.077,335.091,-101.394,174.278,33.490,156.175
C02626=1066.084,335.339,-101.429,174.282,33.494,156.176
C02627=1066.090,335.586,-101.463,174.286,33.499,156.177
C02628=1066.097,335.833,-101.499,174.289,33.504,156.178
C02629=1066.102,336.082,-101.534,174.293,33.509,156.179
C02630=1066.109,336.329,-101.569,174.296,33.514,156.180
C02631=1066.115,336.576,-101.603,174.300,33.519,156.181
C02632=1066.122,336.824,-101.638,174.303,33.524,156.182
C02633=1066.129,337.071,-101.673,174.307,33.528,156.183
C02634=1066.135,337.319,-101.707,174.310,33.534,156.184
C02635=1066.142,337.566,-101.743,174.315,33.538,156.185
C02636=1066.149,337.814,-101.778,174.318,33.544,156.186
C02637=1066.154,338.061,-101.813,174.321,33.549,156.187
C02638=1066.160,338.309,-101.847,174.325,33.554,156.188
C02639=1066.167,338.556,-101.883,174.328,33.559,156.189
C02640=1066.173,338.804,-101.918,174.332,33.564,156.190
C02641=1066.180,339.051,-101.953,174.335,33.569,156.191
C02642=1066.187,339.299,-101.989,174.339,33.574,156.192
C02643=1066.194,339.546,-102.024,174.343,33.579,156.193
C02644=1066.199,339.794,-102.058,174.347,33.584,156.194
C02645=1066.205,340.041,-102.093,174.350,33.589,156.195
C02646=1066.212,340.288,-102.129,174.354,33.594,156.196
C02647=1066.218,340.536,-102.164,174.357,33.599,156.197
C02648=1066.225,340.783,-102.199,174.361,33.604,156.198
C02649=1066.232,341.031,-102.235,174.365,33.609,156.199
C02650=1066.238,341.278,-102.270,174.368,33.615,156.200
C02651=1066.245,341.526,-102.305,174.373,33.620,156.201
C02652=1066.251,341.773,-102.341,174.376,33.624,156.202
C02653=1066.257,342.021,-102.376,174.380,33.630,156.203
C02654=1066.264,342.268,-102.411,174.383,33.635,156.205
C02655=1066.271,342.515,-102.447,174.387,33.640,156.205
C02656=1066.277,342.763,-102.482,174.390,33.645,156.207
C02657=1066.284,343.011,-102.517,174.394,33.650,156.208
C02658=1066.291,343.257,-102.553,174.398,33.655,156.209
C02659=1066.297,343.505,-102.589,174.402,33.661,156.210
C02660=1066.304,343.752,-102.624,174.406,33.665,156.211
C02661=1066.310,344.000,-102.660,174.409,33.671,156.212
C02662=1066.316,344.247,-102.695,174.413,33.676,156.213
C02663=1066.323,344.494,-102.732,174.416,33.681,156.214
C02664=1066.328,344.724,-102.764,174.420,33.686,156.215
C02665=1066.334,344.955,-102.798,174.424,33.691,156.216
C02666=1066.341,345.185,-102.831,174.427,33.696,156.217
C02667=1066.346,345.415,-102.864,174.431,33.701,156.218
C02668=1066.353,345.645,-102.898,174.434,33.706,156.219
C02669=1066.359,345.876,-102.931,174.437,33.711,156.220
C02670=1066.364,346.106,-102.964,174.441,33.716,156.221
C02671=1066.371,346.336,-102.997,174.444,33.720,156.222
C02672=1066.378,346.583,-103.033,174.449,33.725,156.223
C02673=1066.384,346.831,-103.069,174.452,33.731,156.224
C02674=1066.391,347.077,-103.104,174.456,33.736,156.225
C02675=1066.397,347.325,-103.140,174.460,33.742,156.227
C02676=1066.403,347.572,-103.177,174.463,33.747,156.228
C02677=1066.410,347.819,-103.212,174.467,33.752,156.229
C02678=1066.417,348.067,-103.249,174.471,33.757,156.230
C02679=1066.423,348.315,-103.284,174.475,33.763,156.231
C02680=1066.430,348.562,-103.320,174.479,33.768,156.232
C02681=1066.436,348.809,-103.357,174.482,33.774,156.233
C02682=1066.442,349.056,-103.392,174.486,33.779,156.234
C02683=1066.449,349.303,-103.428,174.490,33.784,156.235
C02684=1066.456,349.551,-103.465,174.494,33.790,156.237
C02685=1066.462,349.799,-103.501,174.498,33.795,156.238
C02686=1066.469,350.046,-103.537,174.502,33.800,156.239
C02687=1066.476,350.292,-103.573,174.505,33.806,156.240
C02688=1066.482,350.540,-103.609,174.509,33.811,156.241
C02689=1066.489,350.788,-103.646,174.514,33.817,156.242
C02690=1066.496,351.035,-103.681,174.517,33.822,156.243
C02691=1066.502,351.282,-103.718,174.521,33.828,156.244
C02692=1066.508,351.529,-103.754,174.525,33.833,156.246
C02693=1066.515,351.777,-103.790,174.528,33.839,156.247
C02694=1066.522,352.024,-103.827,174.533,33.844,156.248
C02695=1066.529,352.271,-103.863,174.537,33.850,156.249
C02696=1066.535,352.518,-103.899,174.541,33.855,156.250
C02697=1066.542,352.766,-103.936,174.544,33.861,156.251
C02698=1066.548,353.013,-103.972,174.548,33.866,156.252
C02699=1066.555,353.260,-104.009,174.553,33.872,156.254
C02700=1066.561,353.507,-104.046,174.556,33.877,156.255
C02701=1066.568,353.755,-104.082,174.560,33.883,156.256
C02702=1066.574,354.002,-104.119,174.564,33.888,156.257
C02703=1066.581,354.249,-104.155,174.568,33.894,156.258
C02704=1066.587,354.496,-104.192,174.572,33.899,156.259
C02705=1066.594,354.743,-104.228,174.576,33.905,156.261
C02706=1066.601,354.991,-104.265,174.580,33.910,156.262
C02707=1066.607,355.238,-104.301,174.584,33.916,156.263
C02708=1066.614,355.485,-104.339,174.587,33.922,156.264
C02709=1066.621,355.732,-104.375,174.592,33.927,156.265
C02710=1066.627,355.979,-104.412,174.596,33.933,156.267
C02711=1066.633,356.227,-104.448,174.600,33.939,156.268
C02712=1066.640,356.474,-104.485,174.603,33.944,156.269
C02713=1066.647,356.721,-104.522,174.608,33.950,156.270
C02714=1066.654,356.969,-104.559,174.612,33.955,156.271
C02715=1066.660,357.216,-104.596,174.616,33.961,156.272
C02716=1066.667,357.463,-104.633,174.619,33.967,156.274
C02717=1066.674,357.710,-104.670,174.623,33.972,156.275
C02718=1066.681,357.958,-104.706,174.628,33.978,156.276
C02719=1066.687,358.204,-104.744,174.632,33.984,156.277
C02720=1066.694,358.436,-104.778,174.635,33.989,156.278
C02721=1066.700,358.668,-104.812,174.639,33.994,156.280
C02722=1066.706,358.900,-104.847,174.644,34.000,156.281
C02723=1066.713,359.133,-104.882,174.647,34.005,156.282
C02724=1066.719,359.364,-104.917,174.651,34.011,156.283
C02725=1066.725,359.596,-104.952,174.654,34.016,156.284
C02726=1066.731,359.829,-104.987,174.659,34.022,156.285
C02727=1066.737,360.061,-105.022,174.663,34.027,156.286
C02728=1066.744,360.308,-105.059,174.666,34.033,156.288
C02729=1066.751,360.555,-105.096,174.670,34.039,156.289
C02730=1066.758,360.802,-105.133,174.675,34.045,156.290
C02731=1066.764,361.049,-105.171,174.679,34.051,156.292
C02732=1066.771,361.297,-105.208,174.683,34.056,156.293
C02733=1066.778,361.544,-105.245,174.687,34.062,156.294
C02734=1066.785,361.791,-105.283,174.691,34.068,156.295
C02735=1066.791,362.038,-105.319,174.695,34.074,156.297
C02736=1066.798,362.285,-105.357,174.699,34.080,156.298
C02737=1066.805,362.532,-105.395,174.703,34.085,156.299
C02738=1066.812,362.779,-105.432,174.708,34.092,156.300
C02739=1066.818,363.026,-105.470,174.712,34.097,156.302
C02740=1066.825,363.273,-105.507,174.716,34.104,156.303
C02741=1066.832,363.520,-105.544,174.720,34.110,156.304
C02742=1066.839,363.768,-105.581,174.724,34.115,156.305
C02743=1066.845,364.014,-105.619,174.728,34.121,156.307
C02744=1066.852,364.261,-105.657,174.732,34.127,156.308
C02745=1066.859,364.509,-105.694,174.737,34.133,156.309
C02746=1066.865,364.755,-105.732,174.741,34.139,156.310
C02747=1066.872,365.002,-105.770,174.745,34.145,156.312
C02748=1066.879,365.250,-105.808,174.749,34.152,156.313
C02749=1066.886,365.496,-105.845,174.754,34.157,156.314
C02750=1066.892,365.744,-105.883,174.758,34.164,156.316
C02751=1066.899,365.991,-105.921,174.762,34.170,156.317
C02752=1066.906,366.237,-105.959,174.767,34.176,156.318
C02753=1066.912,366.484,-105.997,174.770,34.182,156.320
C02754=1066.919,366.732,-106.035,174.774,34.188,156.321
C02755=1066.926,366.979,-106.073,174.779,34.194,156.322
C02756=1066.932,367.225,-106.110,174.783,34.201,156.324
C02757=1066.939,367.472,-106.149,174.787,34.207,156.325
C02758=1066.947,367.719,-106.186,174.792,34.213,156.326
C02759=1066.953,367.967,-106.224,174.796,34.219,156.328
C02760=1066.959,368.214,-106.262,174.800,34.225,156.329
C02761=1066.967,368.460,-106.300,174.804,34.231,156.330
C02762=1066.973,368.708,-106.338,174.809,34.238,156.332
C02763=1066.980,368.955,-106.376,174.813,34.244,156.333
C02764=1066.987,369.202,-106.415,174.817,34.250,156.334
C02765=1066.994,369.449,-106.452,174.822,34.256,156.336
C02766=1067.001,369.695,-106.491,174.826,34.263,156.337
C02767=1067.007,369.942,-106.529,174.830,34.269,156.339
C02768=1067.015,370.189,-106.567,174.835,34.275,156.340
C02769=1067.021,370.436,-106.605,174.839,34.281,156.341
C02770=1067.028,370.683,-106.644,174.843,34.288,156.343
C02771=1067.035,370.930,-106.682,174.848,34.294,156.344
C02772=1067.042,371.177,-106.721,174.852,34.301,156.345
C02773=1067.049,371.424,-106.758,174.857,34.307,156.347
C02774=1067.056,371.671,-106.797,174.861,34.313,156.348
C02775=1067.063,371.918,-106.836,174.865,34.319,156.350
C02776=1067.069,372.159,-106.872,174.870,34.326,156.351
C02777=1067.076,372.399,-106.910,174.874,34.332,156.352
C02778=1067.083,372.640,-106.948,174.878,34.338,156.354
C02779=1067.090,372.880,-106.985,174.883,34.344,156.355
C02780=1067.097,373.121,-107.022,174.887,34.350,156.356
C02781=1067.103,373.362,-107.061,174.891,34.357,156.358
C02782=1067.110,373.603,-107.098,174.896,34.363,156.359
C02783=1067.117,373.844,-107.136,174.900,34.370,156.361
C02784=1067.123,374.091,-107.174,174.904,34.376,156.362
C02785=1067.130,374.338,-107.213,174.909,34.383,156.363
C02786=1067.137,374.585,-107.252,174.913,34.389,156.365
C02787=1067.143,374.831,-107.291,174.918,34.396,156.366
C02788=1067.150,375.078,-107.330,174.922,34.402,156.368
C02789=1067.157,375.325,-107.368,174.926,34.409,156.369
C02790=1067.164,375.572,-107.407,174.932,34.416,156.371
C02791=1067.171,375.819,-107.446,174.936,34.422,156.372
C02792=1067.178,376.065,-107.484,174.941,34.429,156.374
C02793=1067.185,376.312,-107.523,174.945,34.436,156.375
C02794=1067.192,376.558,-107.563,174.949,34.442,156.377
C02795=1067.199,376.805,-107.602,174.954,34.449,156.378
C02796=1067.206,377.052,-107.640,174.958,34.455,156.379
C02797=1067.213,377.299,-107.680,174.963,34.462,156.381
C02798=1067.220,377.546,-107.718,174.968,34.469,156.382
C02799=1067.227,377.793,-107.757,174.972,34.476,156.384
C02800=1067.234,378.039,-107.797,174.977,34.482,156.385
C02801=1067.241,378.286,-107.836,174.981,34.489,156.387
C02802=1067.248,378.533,-107.874,174.986,34.496,156.388
C02803=1067.255,378.780,-107.914,174.990,34.502,156.390
C02804=1067.262,379.027,-107.953,174.996,34.509,156.391
C02805=1067.269,379.274,-107.992,175.000,34.516,156.393
C02806=1067.276,379.520,-108.032,175.004,34.523,156.394
C02807=1067.283,379.767,-108.070,175.009,34.530,156.396
C02808=1067.291,380.013,-108.110,175.013,34.537,156.398
C02809=1067.297,380.260,-108.149,175.019,34.543,156.399
C02810=1067.305,380.506,-108.189,175.023,34.550,156.401
C02811=1067.311,380.754,-108.229,175.028,34.557,156.402
C02812=1067.318,381.001,-108.268,175.032,34.564,156.404
C02813=1067.325,381.247,-108.307,175.037,34.571,156.405
C02814=1067.332,381.494,-108.347,175.042,34.578,156.407
C02815=1067.340,381.741,-108.386,175.047,34.585,156.408
C02816=1067.346,381.988,-108.426,175.051,34.592,156.410
C02817=1067.353,382.234,-108.465,175.055,34.599,156.411
C02818=1067.360,382.481,-108.504,175.061,34.606,156.413
C02819=1067.367,382.728,-108.545,175.065,34.613,156.415
C02820=1067.374,382.974,-108.584,175.070,34.620,156.416
C02821=1067.381,383.220,-108.624,175.074,34.627,156.418
C02822=1067.388,383.467,-108.664,175.080,34.634,156.419
C02823=1067.395,383.714,-108.703,175.084,34.641,156.421
C02824=1067.402,383.960,-108.743,175.089,34.648,156.423
C02825=1067.409,384.208,-108.783,175.093,34.656,156.424
C02826=1067.416,384.454,-108.823,175.099,34.663,156.426
C02827=1067.424,384.701,-108.863,175.103,34.670,156.427
C02828=1067.430,384.947,-108.903,175.108,34.677,156.429
C02829=1067.437,385.194,-108.942,175.113,34.684,156.431
C02830=1067.445,385.440,-108.982,175.118,34.691,156.432
C02831=1067.452,385.687,-109.023,175.122,34.699,156.434
C02832=1067.460,385.952,-109.065,175.128,34.706,156.436
C02833=1067.467,386.217,-109.109,175.134,34.714,156.437
C02834=1067.475,386.482,-109.152,175.138,34.722,156.439
C02835=1067.483,386.746,-109.195,175.144,34.730,156.441
C02836=1067.490,386.994,-109.235,175.148,34.738,156.443
C02837=1067.497,387.240,-109.275,175.154,34.745,156.444
C02838=1067.505,387.487,-109.315,175.158,34.752,156.446
C02839=1067.511,387.733,-109.356,175.163,34.759,156.448
C02840=1067.519,387.980,-109.396,175.168,34.766,156.449
C02841=1067.525,388.226,-109.436,175.173,34.774,156.451
C02842=1067.533,388.472,-109.476,175.179,34.781,156.453
C02843=1067.540,388.720,-109.517,175.183,34.789,156.454
C02844=1067.547,388.966,-109.556,175.188,34.796,156.456
C02845=1067.555,389.212,-109.598,175.193,34.804,156.458
C02846=1067.562,389.459,-109.637,175.198,34.811,156.459
C02847=1067.569,389.705,-109.678,175.203,34.819,156.461
C02848=1067.577,389.952,-109.718,175.208,34.826,156.463
C02849=1067.584,390.198,-109.759,175.213,34.834,156.464
C02850=1067.591,390.445,-109.799,175.218,34.841,156.466
C02851=1067.599,390.691,-109.840,175.223,34.848,156.468
C02852=1067.606,390.938,-109.880,175.228,34.856,156.470
C02853=1067.613,391.184,-109.921,175.233,34.864,156.471
C02854=1067.621,391.431,-109.962,175.239,34.872,156.473
C02855=1067.628,391.678,-110.002,175.243,34.879,156.475
C02856=1067.635,391.924,-110.043,175.249,34.887,156.477
C02857=1067.642,392.170,-110.084,175.253,34.894,156.478
C02858=1067.650,392.417,-110.125,175.259,34.902,156.480
C02859=1067.656,392.663,-110.165,175.264,34.910,156.482
C02860=1067.664,392.910,-110.206,175.269,34.918,156.484
C02861=1067.672,393.156,-110.247,175.274,34.926,156.486
C02862=1067.679,393.403,-110.288,175.280,34.934,156.487
C02863=1067.686,393.649,-110.330,175.284,34.941,156.489
C02864=1067.693,393.895,-110.370,175.290,34.949,156.491
C02865=1067.700,394.142,-110.412,175.294,34.957,156.493
C02866=1067.708,394.388,-110.453,175.300,34.965,156.495
C02867=1067.716,394.635,-110.493,175.305,34.973,156.496
C02868=1067.723,394.881,-110.535,175.310,34.980,156.498
C02869=1067.730,395.128,-110.576,175.315,34.989,156.500
C02870=1067.737,395.374,-110.617,175.321,34.996,156.502
C02871=1067.744,395.620,-110.658,175.325,35.004,156.504
C02872=1067.751,395.867,-110.699,175.331,35.012,156.506
C02873=1067.759,396.113,-110.740,175.337,35.020,156.507
C02874=1067.766,396.359,-110.782,175.342,35.029,156.509
C02875=1067.774,396.606,-110.824,175.347,35.036,156.511
C02876=1067.781,396.853,-110.865,175.352,35.045,156.513
C02877=1067.788,397.099,-110.906,175.358,35.053,156.515
C02878=1067.796,397.345,-110.948,175.362,35.061,156.517
C02879=1067.803,397.592,-110.989,175.368,35.069,156.519
C02880=1067.811,397.838,-111.030,175.374,35.077,156.521
C02881=1067.818,398.084,-111.072,175.378,35.085,156.522
C02882=1067.825,398.331,-111.114,175.384,35.093,156.524
C02883=1067.833,398.577,-111.156,175.390,35.102,156.526
C02884=1067.840,398.823,-111.197,175.395,35.110,156.528
C02885=1067.848,399.069,-111.239,175.400,35.118,156.530
C02886=1067.855,399.316,-111.280,175.405,35.126,156.532
C02887=1067.863,399.563,-111.322,175.411,35.135,156.534
C02888=1067.871,399.844,-111.370,175.417,35.144,156.536
C02889=1067.879,400.125,-111.417,175.424,35.154,156.538
C02890=1067.888,400.405,-111.465,175.430,35.163,156.541
C02891=1067.896,400.687,-111.513,175.435,35.173,156.543
C02892=1067.904,400.933,-111.555,175.441,35.181,156.545
C02893=1067.911,401.179,-111.597,175.447,35.190,156.547
C02894=1067.920,401.426,-111.639,175.453,35.198,156.549
C02895=1067.927,401.672,-111.680,175.458,35.207,156.551
C02896=1067.934,401.919,-111.723,175.463,35.215,156.553
C02897=1067.941,402.165,-111.765,175.469,35.224,156.555
C02898=1067.949,402.411,-111.807,175.475,35.232,156.557
C02899=1067.957,402.657,-111.849,175.480,35.241,156.559
C02900=1067.964,402.904,-111.892,175.486,35.250,156.561
C02901=1067.972,403.150,-111.934,175.492,35.258,156.563
C02902=1067.980,403.396,-111.976,175.497,35.266,156.565
C02903=1067.987,403.642,-112.018,175.502,35.275,156.567
C02904=1067.995,403.889,-112.061,175.508,35.284,156.569
C02905=1068.002,404.135,-112.103,175.514,35.293,156.571
C02906=1068.009,404.381,-112.145,175.520,35.302,156.573
C02907=1068.017,404.628,-112.188,175.526,35.310,156.575
C02908=1068.025,404.874,-112.231,175.530,35.319,156.577
C02909=1068.032,405.120,-112.273,175.536,35.328,156.580
C02910=1068.040,405.366,-112.315,175.542,35.337,156.582
C02911=1068.047,405.613,-112.358,175.548,35.346,156.584
C02912=1068.056,405.859,-112.401,175.554,35.354,156.586
C02913=1068.063,406.105,-112.443,175.560,35.364,156.588
C02914=1068.071,406.352,-112.486,175.566,35.372,156.590
C02915=1068.078,406.597,-112.529,175.571,35.381,156.592
C02916=1068.085,406.844,-112.572,175.577,35.390,156.594
C02917=1068.093,407.090,-112.614,175.583,35.399,156.597
C02918=1068.101,407.337,-112.657,175.589,35.409,156.599
C02919=1068.109,407.582,-112.700,175.594,35.418,156.601
C02920=1068.116,407.829,-112.743,175.600,35.427,156.603
C02921=1068.123,408.075,-112.786,175.606,35.436,156.605
C02922=1068.132,408.321,-112.829,175.612,35.445,156.607
C02923=1068.139,408.567,-112.872,175.618,35.454,156.610
C02924=1068.146,408.813,-112.915,175.624,35.463,156.612
C02925=1068.154,409.059,-112.958,175.630,35.472,156.614
C02926=1068.162,409.306,-113.001,175.636,35.482,156.616
C02927=1068.170,409.552,-113.044,175.642,35.491,156.619
C02928=1068.177,409.797,-113.087,175.648,35.500,156.621
C02929=1068.185,410.044,-113.131,175.654,35.510,156.623
C02930=1068.193,410.290,-113.174,175.660,35.519,156.625
C02931=1068.200,410.536,-113.218,175.666,35.528,156.627
C02932=1068.209,410.782,-113.261,175.672,35.538,156.630
C02933=1068.216,411.028,-113.304,175.678,35.547,156.632
C02934=1068.224,411.275,-113.348,175.684,35.556,156.634
C02935=1068.232,411.520,-113.391,175.690,35.566,156.637
C02936=1068.240,411.766,-113.434,175.696,35.576,156.639
C02937=1068.248,412.013,-113.478,175.702,35.585,156.641
C02938=1068.255,412.259,-113.521,175.709,35.595,156.643
C02939=1068.264,412.505,-113.564,175.715,35.604,156.646
C02940=1068.271,412.751,-113.608,175.721,35.614,156.648
C02941=1068.279,412.997,-113.652,175.728,35.623,156.650
C02942=1068.287,413.243,-113.696,175.734,35.633,156.653
C02943=1068.295,413.489,-113.739,175.740,35.642,156.655
C02944=1068.304,413.774,-113.790,175.747,35.654,156.658
C02945=1068.313,414.059,-113.840,175.754,35.665,156.661
C02946=1068.322,414.344,-113.892,175.762,35.676,156.663
C02947=1068.332,414.629,-113.942,175.769,35.687,156.666
C02948=1068.340,414.876,-113.985,175.775,35.698,156.668
C02949=1068.348,415.121,-114.030,175.781,35.707,156.671
C02950=1068.356,415.367,-114.074,175.789,35.717,156.673
C02951=1068.363,415.614,-114.118,175.795,35.727,156.676
C02952=1068.372,415.859,-114.162,175.801,35.737,156.678
C02953=1068.379,416.106,-114.206,175.807,35.747,156.681
C02954=1068.387,416.351,-114.250,175.814,35.758,156.683
C02955=1068.395,416.597,-114.294,175.820,35.767,156.685
C02956=1068.403,416.843,-114.339,175.827,35.777,156.688
C02957=1068.411,417.089,-114.384,175.833,35.787,156.690
C02958=1068.419,417.335,-114.427,175.840,35.798,156.693
C02959=1068.427,417.581,-114.472,175.846,35.808,156.695
C02960=1068.435,417.827,-114.516,175.853,35.818,156.698
C02961=1068.443,418.073,-114.561,175.860,35.829,156.701
C02962=1068.451,418.319,-114.605,175.866,35.839,156.703
C02963=1068.460,418.565,-114.649,175.872,35.849,156.706
C02964=1068.468,418.810,-114.694,175.880,35.859,156.708
C02965=1068.475,419.057,-114.739,175.886,35.870,156.711
C02966=1068.484,419.303,-114.783,175.893,35.880,156.713
C02967=1068.492,419.548,-114.828,175.899,35.890,156.716
C02968=1068.500,419.794,-114.873,175.906,35.900,156.718
C02969=1068.508,420.040,-114.917,175.913,35.911,156.721
C02970=1068.517,420.286,-114.962,175.919,35.922,156.724
C02971=1068.524,420.531,-115.007,175.927,35.932,156.726
C02972=1068.532,420.777,-115.052,175.933,35.942,156.729
C02973=1068.541,421.024,-115.096,175.940,35.953,156.731
C02974=1068.550,421.269,-115.141,175.947,35.964,156.734
C02975=1068.557,421.515,-115.186,175.954,35.974,156.737
C02976=1068.566,421.761,-115.232,175.961,35.985,156.739
C02977=1068.573,422.007,-115.277,175.968,35.996,156.742
C02978=1068.582,422.252,-115.322,175.974,36.007,156.745
C02979=1068.589,422.499,-115.367,175.982,36.017,156.747
C02980=1068.598,422.744,-115.412,175.988,36.028,156.750
C02981=1068.606,422.989,-115.457,175.996,36.039,156.753
C02982=1068.614,423.236,-115.503,176.002,36.050,156.755
C02983=1068.623,423.481,-115.548,176.009,36.061,156.758
C02984=1068.631,423.727,-115.594,176.017,36.072,156.761
C02985=1068.639,423.972,-115.639,176.023,36.083,156.764
C02986=1068.647,424.218,-115.685,176.031,36.094,156.766
C02987=1068.656,424.463,-115.730,176.038,36.105,156.769
C02988=1068.664,424.709,-115.776,176.045,36.116,156.772
C02989=1068.672,424.955,-115.820,176.052,36.127,156.775
C02990=1068.680,425.201,-115.866,176.060,36.138,156.778
C02991=1068.689,425.446,-115.912,176.066,36.149,156.780
C02992=1068.697,425.692,-115.958,176.074,36.160,156.783
C02993=1068.706,425.938,-116.003,176.081,36.172,156.786
C02994=1068.714,426.183,-116.049,176.088,36.183,156.789
C02995=1068.723,426.429,-116.094,176.096,36.194,156.792
C02996=1068.731,426.675,-116.140,176.103,36.206,156.795
C02997=1068.740,426.920,-116.186,176.111,36.217,156.797
C02998=1068.748,427.166,-116.232,176.117,36.228,156.800
C02999=1068.756,427.412,-116.278,176.125,36.240,156.803
C03000=1068.767,427.716,-116.335,176.134,36.254,156.807
C03001=1068.777,428.020,-116.392,176.144,36.268,156.810
C03002=1068.788,428.324,-116.450,176.153,36.283,156.814
C03003=1068.798,428.629,-116.507,176.162,36.297,156.818
C03004=1068.807,428.875,-116.553,176.170,36.309,156.821
C03005=1068.815,429.120,-116.599,176.177,36.321,156.824
C03006=1068.824,429.366,-116.646,176.185,36.332,156.827
C03007=1068.832,429.611,-116.691,176.193,36.344,156.830
C03008=1068.841,429.856,-116.738,176.201,36.356,156.833
C03009=1068.849,430.102,-116.785,176.208,36.368,156.836
C03010=1068.858,430.347,-116.831,176.215,36.379,156.839
C03011=1068.867,430.593,-116.878,176.223,36.391,156.842
C03012=1068.875,430.838,-116.924,176.231,36.403,156.845
C03013=1068.884,431.084,-116.971,176.238,36.415,156.848
C03014=1068.893,431.329,-117.018,176.246,36.427,156.851
C03015=1068.901,431.575,-117.064,176.254,36.439,156.854
C03016=1068.910,431.820,-117.111,176.262,36.451,156.857
C03017=1068.918,432.066,-117.158,176.270,36.464,156.860
C03018=1068.927,432.311,-117.205,176.278,36.476,156.863
C03019=1068.935,432.557,-117.251,176.286,36.488,156.867
C03020=1068.944,432.802,-117.299,176.294,36.500,156.870
C03021=1068.953,433.047,-117.346,176.302,36.513,156.873
C03022=1068.961,433.293,-117.392,176.310,36.525,156.876
C03023=1068.970,433.537,-117.440,176.318,36.538,156.879
C03024=1068.979,433.783,-117.486,176.326,36.550,156.883
C03025=1068.987,434.028,-117.534,176.334,36.562,156.886
C03026=1068.995,434.274,-117.581,176.342,36.575,156.889
C03027=1069.005,434.519,-117.629,176.351,36.588,156.892
C03028=1069.014,434.764,-117.676,176.359,36.600,156.896
C03029=1069.022,435.010,-117.723,176.367,36.613,156.899
C03030=1069.031,435.255,-117.771,176.375,36.626,156.902
C03031=1069.040,435.499,-117.818,176.383,36.638,156.905
C03032=1069.049,435.746,-117.865,176.392,36.651,156.909
C03033=1069.058,435.991,-117.913,176.400,36.663,156.912
C03034=1069.066,436.236,-117.961,176.408,36.676,156.915
C03035=1069.075,436.481,-118.008,176.417,36.689,156.919
C03036=1069.084,436.726,-118.056,176.425,36.702,156.922
C03037=1069.093,436.971,-118.103,176.433,36.715,156.926
C03038=1069.103,437.217,-118.151,176.442,36.728,156.929
C03039=1069.111,437.462,-118.199,176.451,36.741,156.932
C03040=1069.121,437.707,-118.246,176.459,36.754,156.936
C03041=1069.129,437.952,-118.295,176.468,36.767,156.939
C03042=1069.139,438.197,-118.343,176.476,36.780,156.943
C03043=1069.148,438.442,-118.390,176.485,36.793,156.946
C03044=1069.157,438.688,-118.438,176.493,36.807,156.950
C03045=1069.165,438.933,-118.487,176.502,36.820,156.953
C03046=1069.175,439.178,-118.535,176.511,36.833,156.957
C03047=1069.184,439.422,-118.583,176.519,36.847,156.960
C03048=1069.193,439.668,-118.631,176.529,36.860,156.964
C03049=1069.202,439.913,-118.680,176.537,36.874,156.967
C03050=1069.211,440.158,-118.728,176.546,36.887,156.971
C03051=1069.220,440.403,-118.776,176.555,36.901,156.975
C03052=1069.230,440.648,-118.825,176.564,36.914,156.978
C03053=1069.238,440.894,-118.873,176.573,36.928,156.982
C03054=1069.247,441.138,-118.921,176.582,36.941,156.985
C03055=1069.257,441.383,-118.970,176.591,36.955,156.989
C03056=1069.269,441.724,-119.038,176.603,36.975,156.994
C03057=1069.283,442.065,-119.106,176.616,36.994,156.999
C03058=1069.295,442.407,-119.174,176.629,37.013,157.004
C03059=1069.308,442.748,-119.243,176.642,37.033,157.010
C03060=1069.318,442.993,-119.291,176.651,37.047,157.014
C03061=1069.327,443.238,-119.340,176.661,37.061,157.017
C03062=1069.336,443.483,-119.389,176.669,37.075,157.021
C03063=1069.345,443.727,-119.438,176.679,37.089,157.025
C03064=1069.354,443.973,-119.487,176.688,37.103,157.029
C03065=1069.364,444.218,-119.536,176.698,37.117,157.032
C03066=1069.373,444.462,-119.586,176.708,37.132,157.036
C03067=1069.382,444.707,-119.635,176.716,37.146,157.040
C03068=1069.392,444.952,-119.684,176.726,37.161,157.044
C03069=1069.402,445.196,-119.734,176.736,37.175,157.048
C03070=1069.411,445.442,-119.783,176.745,37.190,157.052
C03071=1069.420,445.686,-119.833,176.755,37.205,157.056
C03072=1069.430,445.931,-119.882,176.765,37.219,157.060
C03073=1069.439,446.175,-119.932,176.775,37.233,157.064
C03074=1069.449,446.421,-119.981,176.784,37.248,157.068
C03075=1069.458,446.666,-120.031,176.794,37.263,157.072
C03076=1069.470,446.961,-120.092,176.807,37.281,157.077
C03077=1069.481,447.256,-120.152,176.818,37.299,157.082
C03078=1069.493,447.551,-120.211,176.831,37.317,157.087
C03079=1069.505,447.846,-120.272,176.842,37.335,157.092
C03080=1069.514,448.090,-120.321,176.852,37.350,157.096
C03081=1069.525,448.333,-120.370,176.862,37.365,157.100
C03082=1069.536,448.578,-120.419,176.872,37.379,157.104
C03083=1069.548,448.823,-120.468,176.880,37.393,157.107
C03084=1069.562,449.068,-120.515,176.889,37.406,157.111
C03085=1069.577,449.312,-120.561,176.899,37.419,157.115
C03086=1069.593,449.558,-120.607,176.906,37.432,157.118
C03087=1069.610,449.803,-120.653,176.915,37.445,157.122
C03088=1069.263,449.804,-120.908,176.902,37.581,157.158
C03089=1069.247,449.559,-120.862,176.894,37.569,157.155
C03090=1069.230,449.313,-120.816,176.885,37.556,157.151
C03091=1069.216,449.068,-120.769,176.877,37.544,157.148
C03092=1069.201,448.824,-120.722,176.867,37.530,157.144
C03093=1069.189,448.579,-120.675,176.858,37.516,157.140
C03094=1069.177,448.334,-120.626,176.848,37.502,157.136
C03095=1069.166,448.091,-120.576,176.838,37.487,157.132
C03096=1069.156,447.848,-120.527,176.828,37.472,157.128
C03097=1069.147,447.603,-120.477,176.818,37.457,157.124
C03098=1069.137,447.358,-120.427,176.808,37.442,157.120
C03099=1069.128,447.113,-120.377,176.797,37.427,157.116
C03100=1069.118,446.869,-120.327,176.787,37.413,157.112
C03101=1069.108,446.624,-120.278,176.778,37.398,157.108
C03102=1069.099,446.379,-120.228,176.768,37.383,157.104
C03103=1069.089,446.134,-120.178,176.758,37.368,157.100
C03104=1069.080,445.889,-120.128,176.748,37.354,157.096
C03105=1069.070,445.645,-120.079,176.738,37.339,157.092
C03106=1069.060,445.400,-120.029,176.728,37.325,157.088
C03107=1069.051,445.156,-119.979,176.719,37.310,157.084
C03108=1069.042,444.911,-119.930,176.710,37.296,157.080
C03109=1069.032,444.666,-119.881,176.700,37.281,157.076
C03110=1069.023,444.421,-119.831,176.690,37.267,157.072
C03111=1069.014,444.176,-119.782,176.681,37.253,157.068
C03112=1069.005,443.931,-119.732,176.671,37.239,157.064
C03113=1068.995,443.687,-119.683,176.661,37.224,157.061
C03114=1068.986,443.441,-119.634,176.652,37.210,157.057
C03115=1068.976,443.196,-119.586,176.643,37.196,157.053
C03116=1068.966,442.952,-119.536,176.633,37.182,157.049
C03117=1068.953,442.578,-119.462,176.619,37.160,157.043
C03118=1068.938,442.205,-119.387,176.605,37.140,157.038
C03119=1068.924,441.832,-119.313,176.591,37.119,157.032
C03120=1068.910,441.460,-119.238,176.577,37.098,157.026
C03121=1068.901,441.215,-119.190,176.567,37.084,157.023
C03122=1068.892,440.970,-119.141,176.559,37.070,157.019
C03123=1068.882,440.725,-119.092,176.550,37.057,157.015
C03124=1068.874,440.480,-119.045,176.541,37.043,157.012
C03125=1068.865,440.235,-118.995,176.532,37.029,157.008
C03126=1068.855,439.990,-118.947,176.522,37.016,157.005
C03127=1068.846,439.745,-118.899,176.514,37.002,157.001
C03128=1068.837,439.500,-118.850,176.504,36.989,156.997
C03129=1068.824,439.155,-118.783,176.492,36.970,156.992
C03130=1068.811,438.811,-118.715,176.480,36.951,156.987
C03131=1068.799,438.467,-118.647,176.468,36.933,156.982
C03132=1068.786,438.122,-118.580,176.456,36.915,156.978
C03133=1068.777,437.877,-118.532,176.447,36.901,156.974
C03134=1068.767,437.632,-118.484,176.438,36.888,156.971
C03135=1068.758,437.388,-118.436,176.430,36.875,156.967
C03136=1068.750,437.142,-118.388,176.421,36.862,156.964
C03137=1068.741,436.897,-118.341,176.412,36.850,156.961
C03138=1068.731,436.651,-118.293,176.404,36.837,156.957
C03139=1068.723,436.406,-118.245,176.395,36.824,156.954
C03140=1068.714,436.161,-118.198,176.387,36.811,156.950
C03141=1068.704,435.916,-118.150,176.379,36.798,156.947
C03142=1068.695,435.671,-118.103,176.371,36.785,156.944
C03143=1068.687,435.426,-118.055,176.362,36.772,156.940
C03144=1068.678,435.180,-118.007,176.354,36.760,156.937
C03145=1068.669,434.935,-117.960,176.345,36.748,156.934
C03146=1068.660,434.690,-117.913,176.337,36.735,156.930
C03147=1068.652,434.445,-117.865,176.328,36.722,156.927
C03148=1068.642,434.199,-117.818,176.320,36.710,156.924
C03149=1068.634,433.954,-117.771,176.312,36.697,156.921
C03150=1068.625,433.709,-117.723,176.304,36.685,156.917
C03151=1068.616,433.463,-117.676,176.296,36.672,156.914
C03152=1068.607,433.218,-117.629,176.288,36.660,156.911
C03153=1068.599,432.973,-117.582,176.280,36.648,156.908
C03154=1068.590,432.727,-117.536,176.271,36.635,156.905
C03155=1068.582,432.482,-117.488,176.263,36.623,156.902
C03156=1068.574,432.237,-117.441,176.255,36.611,156.898
C03157=1068.565,431.991,-117.394,176.248,36.599,156.895
C03158=1068.557,431.746,-117.347,176.240,36.586,156.892
C03159=1068.548,431.501,-117.300,176.232,36.574,156.889
C03160=1068.539,431.255,-117.253,176.224,36.562,156.886
C03161=1068.530,431.010,-117.207,176.216,36.550,156.883
C03162=1068.521,430.765,-117.160,176.208,36.538,156.880
C03163=1068.513,430.519,-117.114,176.200,36.526,156.877
C03164=1068.504,430.274,-117.067,176.193,36.515,156.874
C03165=1068.496,430.028,-117.020,176.185,36.503,156.870
C03166=1068.487,429.782,-116.975,176.177,36.491,156.868
C03167=1068.478,429.537,-116.928,176.169,36.479,156.864
C03168=1068.470,429.291,-116.881,176.162,36.468,156.861
C03169=1068.462,429.065,-116.839,176.155,36.457,156.859
C03170=1068.454,428.839,-116.796,176.148,36.446,156.856
C03171=1068.446,428.613,-116.753,176.140,36.435,156.853
C03172=1068.438,428.387,-116.711,176.134,36.425,156.850
C03173=1068.431,428.161,-116.668,176.127,36.414,156.848
C03174=1068.423,427.934,-116.625,176.120,36.403,156.845
C03175=1068.415,427.708,-116.583,176.113,36.393,156.842
C03176=1068.407,427.482,-116.540,176.106,36.382,156.840
C03177=1068.399,427.236,-116.494,176.099,36.371,156.837
C03178=1068.390,426.990,-116.449,176.091,36.359,156.834
C03179=1068.382,426.745,-116.402,176.084,36.348,156.831
C03180=1068.373,426.499,-116.357,176.076,36.337,156.828
C03181=1068.365,426.253,-116.311,176.069,36.326,156.825
C03182=1068.356,426.008,-116.265,176.062,36.314,156.822
C03183=1068.348,425.763,-116.219,176.054,36.303,156.820
C03184=1068.339,425.517,-116.174,176.047,36.292,156.817
C03185=1068.331,425.271,-116.128,176.040,36.280,156.814
C03186=1068.322,425.026,-116.083,176.032,36.269,156.811
C03187=1068.314,424.780,-116.037,176.025,36.258,156.808
C03188=1068.306,424.534,-115.992,176.018,36.247,156.805
C03189=1068.298,424.288,-115.946,176.011,36.237,156.803
C03190=1068.289,424.043,-115.901,176.003,36.226,156.800
C03191=1068.281,423.797,-115.855,175.997,36.215,156.797
C03192=1068.273,423.552,-115.809,175.989,36.203,156.794
C03193=1068.264,423.306,-115.763,175.982,36.193,156.792
C03194=1068.256,423.060,-115.719,175.975,36.182,156.789
C03195=1068.248,422.814,-115.673,175.968,36.171,156.786
C03196=1068.240,422.569,-115.628,175.961,36.160,156.783
C03197=1068.231,422.324,-115.583,175.954,36.149,156.781
C03198=1068.223,422.077,-115.538,175.947,36.138,156.778
C03199=1068.215,421.832,-115.493,175.940,36.128,156.775
C03200=1068.207,421.585,-115.447,175.933,36.117,156.773
C03201=1068.199,421.340,-115.402,175.926,36.107,156.770
C03202=1068.191,421.094,-115.357,175.919,36.096,156.767
C03203=1068.182,420.848,-115.312,175.912,36.085,156.765
C03204=1068.174,420.602,-115.268,175.906,36.075,156.762
C03205=1068.166,420.357,-115.223,175.898,36.064,156.760
C03206=1068.157,420.111,-115.178,175.892,36.054,156.757
C03207=1068.150,419.865,-115.133,175.884,36.043,156.754
C03208=1068.142,419.619,-115.089,175.878,36.033,156.752
C03209=1068.133,419.374,-115.044,175.871,36.023,156.749
C03210=1068.125,419.127,-114.999,175.864,36.012,156.747
C03211=1068.117,418.882,-114.955,175.858,36.002,156.744
C03212=1068.109,418.636,-114.910,175.851,35.992,156.742
C03213=1068.101,418.390,-114.866,175.844,35.981,156.739
C03214=1068.093,418.143,-114.821,175.838,35.971,156.736
C03215=1068.085,417.898,-114.776,175.831,35.961,156.734
C03216=1068.076,417.652,-114.732,175.825,35.951,156.731
C03217=1068.068,417.406,-114.688,175.818,35.941,156.729
C03218=1068.060,417.160,-114.643,175.811,35.931,156.726
C03219=1068.052,416.915,-114.599,175.805,35.921,156.724
C03220=1068.044,416.669,-114.555,175.798,35.910,156.721
C03221=1068.036,416.423,-114.510,175.791,35.900,156.719
C03222=1068.028,416.177,-114.467,175.785,35.890,156.716
C03223=1068.021,415.931,-114.422,175.779,35.880,156.714
C03224=1068.013,415.685,-114.377,175.772,35.870,156.712
C03225=1068.005,415.439,-114.334,175.765,35.860,156.709
C03226=1067.997,415.193,-114.289,175.759,35.851,156.707
C03227=1067.989,414.947,-114.245,175.753,35.840,156.704
C03228=1067.981,414.701,-114.201,175.747,35.831,156.702
C03229=1067.971,414.414,-114.150,175.739,35.820,156.699
C03230=1067.962,414.127,-114.099,175.732,35.808,156.696
C03231=1067.953,413.840,-114.048,175.724,35.797,156.694
C03232=1067.944,413.554,-113.997,175.716,35.785,156.691
C03233=1067.936,413.307,-113.953,175.710,35.776,156.688
C03234=1067.928,413.061,-113.909,175.704,35.766,156.686
C03235=1067.919,412.815,-113.866,175.698,35.756,156.684
C03236=1067.912,412.569,-113.822,175.692,35.747,156.682
C03237=1067.904,412.323,-113.779,175.685,35.738,156.679
C03238=1067.896,412.077,-113.734,175.679,35.728,156.677
C03239=1067.888,411.832,-113.692,175.673,35.718,156.674
C03240=1067.880,411.585,-113.648,175.667,35.709,156.672
C03241=1067.872,411.339,-113.604,175.660,35.699,156.670
C03242=1067.865,411.092,-113.561,175.654,35.690,156.668
C03243=1067.856,410.846,-113.518,175.648,35.681,156.665
C03244=1067.849,410.601,-113.475,175.642,35.671,156.663
C03245=1067.841,410.354,-113.431,175.636,35.662,156.661
C03246=1067.833,410.108,-113.388,175.630,35.653,156.659
C03247=1067.825,409.863,-113.345,175.624,35.643,156.656
C03248=1067.818,409.616,-113.301,175.618,35.634,156.654
C03249=1067.809,409.370,-113.258,175.611,35.625,156.652
C03250=1067.802,409.124,-113.215,175.605,35.615,156.650
C03251=1067.795,408.878,-113.172,175.599,35.606,156.647
C03252=1067.786,408.632,-113.129,175.593,35.597,156.645
C03253=1067.779,408.386,-113.086,175.587,35.588,156.643
C03254=1067.771,408.139,-113.043,175.581,35.579,156.641
C03255=1067.764,407.894,-113.000,175.575,35.569,156.639
C03256=1067.756,407.647,-112.956,175.570,35.561,156.637
C03257=1067.749,407.401,-112.914,175.564,35.552,156.634
C03258=1067.740,407.155,-112.871,175.558,35.542,156.632
C03259=1067.733,406.908,-112.828,175.552,35.533,156.630
C03260=1067.726,406.662,-112.785,175.547,35.525,156.628
C03261=1067.718,406.416,-112.743,175.541,35.515,156.626
C03262=1067.710,406.170,-112.699,175.535,35.506,156.623
C03263=1067.703,405.924,-112.657,175.529,35.498,156.621
C03264=1067.695,405.677,-112.614,175.523,35.489,156.619
C03265=1067.687,405.432,-112.572,175.518,35.480,156.617
C03266=1067.680,405.185,-112.529,175.512,35.471,156.615
C03267=1067.672,404.939,-112.487,175.506,35.462,156.613
C03268=1067.665,404.692,-112.443,175.500,35.453,156.611
C03269=1067.657,404.446,-112.401,175.494,35.444,156.609
C03270=1067.649,404.200,-112.359,175.489,35.436,156.607
C03271=1067.642,403.953,-112.316,175.483,35.427,156.605
C03272=1067.634,403.707,-112.274,175.477,35.418,156.603
C03273=1067.627,403.460,-112.231,175.471,35.410,156.600
C03274=1067.619,403.215,-112.189,175.466,35.401,156.598
C03275=1067.611,402.969,-112.147,175.461,35.392,156.596
C03276=1067.603,402.722,-112.105,175.455,35.384,156.594
C03277=1067.596,402.476,-112.062,175.449,35.375,156.592
C03278=1067.589,402.229,-112.021,175.443,35.367,156.590
C03279=1067.581,401.983,-111.978,175.438,35.359,156.588
C03280=1067.573,401.737,-111.937,175.432,35.350,156.586
C03281=1067.567,401.490,-111.894,175.426,35.341,156.584
C03282=1067.559,401.245,-111.852,175.421,35.333,156.582
C03283=1067.551,400.998,-111.810,175.416,35.325,156.580
C03284=1067.543,400.751,-111.768,175.410,35.316,156.578
C03285=1067.535,400.469,-111.720,175.404,35.306,156.576
C03286=1067.526,400.186,-111.672,175.397,35.297,156.574
C03287=1067.518,399.903,-111.624,175.391,35.287,156.572
C03288=1067.509,399.621,-111.576,175.385,35.278,156.569
C03289=1067.501,399.375,-111.534,175.379,35.270,156.567
C03290=1067.494,399.128,-111.493,175.374,35.261,156.565
C03291=1067.487,398.882,-111.450,175.369,35.253,156.563
C03292=1067.480,398.635,-111.409,175.363,35.245,156.562
C03293=1067.472,398.389,-111.367,175.357,35.236,156.560
C03294=1067.465,398.143,-111.326,175.353,35.228,156.558
C03295=1067.457,397.897,-111.284,175.347,35.220,156.556
C03296=1067.450,397.650,-111.243,175.342,35.212,156.554
C03297=1067.442,397.404,-111.201,175.336,35.204,156.552
C03298=1067.435,397.158,-111.159,175.330,35.196,156.550
C03299=1067.428,396.911,-111.118,175.326,35.188,156.548
C03300=1067.420,396.665,-111.076,175.320,35.179,156.546
C03301=1067.413,396.418,-111.035,175.315,35.172,156.544
C03302=1067.406,396.172,-110.994,175.310,35.163,156.543
C03303=1067.398,395.925,-110.953,175.304,35.156,156.541
C03304=1067.390,395.680,-110.911,175.299,35.148,156.539
C03305=1067.383,395.433,-110.870,175.293,35.140,156.537
C03306=1067.376,395.186,-110.829,175.289,35.132,156.535
C03307=1067.368,394.940,-110.788,175.283,35.124,156.533
C03308=1067.361,394.693,-110.746,175.278,35.116,156.531
C03309=1067.354,394.447,-110.705,175.272,35.108,156.530
C03310=1067.346,394.200,-110.664,175.268,35.100,156.528
C03311=1067.340,393.954,-110.623,175.262,35.092,156.526
C03312=1067.332,393.707,-110.582,175.257,35.084,156.524
C03313=1067.324,393.461,-110.541,175.252,35.077,156.522
C03314=1067.317,393.215,-110.500,175.247,35.069,156.521
C03315=1067.310,392.968,-110.459,175.241,35.061,156.519
C03316=1067.303,392.722,-110.418,175.237,35.054,156.517
C03317=1067.295,392.476,-110.377,175.231,35.046,156.515
C03318=1067.288,392.229,-110.337,175.226,35.038,156.514
C03319=1067.281,391.982,-110.295,175.221,35.030,156.512
C03320=1067.273,391.736,-110.255,175.216,35.023,156.510
C03321=1067.266,391.490,-110.214,175.210,35.015,156.508
C03322=1067.259,391.243,-110.173,175.206,35.007,156.506
C03323=1067.252,390.996,-110.132,175.200,34.999,156.505
C03324=1067.244,390.750,-110.092,175.195,34.992,156.503
C03325=1067.237,390.503,-110.051,175.190,34.984,156.501
C03326=1067.229,390.257,-110.011,175.185,34.977,156.499
C03327=1067.222,390.010,-109.970,175.181,34.970,156.498
C03328=1067.215,389.764,-109.930,175.175,34.962,156.496
C03329=1067.208,389.518,-109.889,175.170,34.955,156.494
C03330=1067.200,389.271,-109.849,175.165,34.947,156.493
C03331=1067.194,389.024,-109.809,175.160,34.940,156.491
C03332=1067.186,388.778,-109.768,175.154,34.932,156.489
C03333=1067.179,388.531,-109.728,175.150,34.925,156.488
C03334=1067.171,388.285,-109.687,175.145,34.918,156.486
C03335=1067.163,388.038,-109.647,175.140,34.910,156.484
C03336=1067.157,387.792,-109.607,175.135,34.903,156.482
C03337=1067.149,387.545,-109.567,175.130,34.895,156.481
C03338=1067.143,387.299,-109.526,175.125,34.888,156.479
C03339=1067.135,387.052,-109.486,175.120,34.881,156.478
C03340=1067.129,386.805,-109.446,175.115,34.873,156.476
C03341=1067.120,386.538,-109.403,175.110,34.865,156.474
C03342=1067.112,386.273,-109.359,175.105,34.858,156.472
C03343=1067.105,386.006,-109.316,175.099,34.850,156.470
C03344=1067.097,385.740,-109.273,175.094,34.842,156.469
C03345=1067.090,385.493,-109.233,175.089,34.835,156.467
C03346=1067.083,385.246,-109.193,175.084,34.828,156.465
C03347=1067.076,384.999,-109.153,175.080,34.820,156.464
C03348=1067.069,384.753,-109.113,175.074,34.813,156.462
C03349=1067.061,384.506,-109.073,175.070,34.806,156.461
C03350=1067.055,384.260,-109.033,175.065,34.799,156.459
C03351=1067.047,384.013,-108.993,175.060,34.792,156.457
C03352=1067.040,383.766,-108.953,175.055,34.785,156.456
C03353=1067.033,383.520,-108.913,175.050,34.778,156.454
C03354=1067.026,383.273,-108.873,175.046,34.770,156.452
C03355=1067.019,383.026,-108.835,175.041,34.764,156.451
C03356=1067.012,382.780,-108.794,175.036,34.756,156.449
C03357=1067.005,382.533,-108.755,175.031,34.750,156.448
C03358=1066.998,382.287,-108.715,175.027,34.742,156.446
C03359=1066.991,382.040,-108.675,175.022,34.735,156.445
C03360=1066.984,381.793,-108.636,175.017,34.728,156.443
C03361=1066.977,381.546,-108.596,175.012,34.721,156.441
C03362=1066.970,381.300,-108.556,175.008,34.714,156.440
C03363=1066.963,381.053,-108.517,175.003,34.707,156.438
C03364=1066.956,380.806,-108.477,174.999,34.701,156.437
C03365=1066.949,380.559,-108.438,174.993,34.694,156.435
C03366=1066.942,380.313,-108.399,174.989,34.687,156.434
C03367=1066.935,380.066,-108.360,174.984,34.680,156.432
C03368=1066.927,379.819,-108.320,174.980,34.673,156.431
C03369=1066.920,379.572,-108.281,174.974,34.666,156.429
C03370=1066.913,379.326,-108.242,174.970,34.660,156.428
C03371=1066.906,379.079,-108.202,174.965,34.653,156.426
C03372=1066.899,378.833,-108.163,174.961,34.646,156.425
C03373=1066.892,378.586,-108.124,174.957,34.639,156.423
C03374=1066.885,378.339,-108.085,174.952,34.633,156.422
C03375=1066.878,378.093,-108.046,174.947,34.626,156.420
C03376=1066.871,377.846,-108.007,174.942,34.619,156.419
C03377=1066.864,377.598,-107.968,174.938,34.612,156.417
C03378=1066.857,377.352,-107.929,174.933,34.606,156.416
C03379=1066.850,377.105,-107.889,174.929,34.599,156.414
C03380=1066.843,376.858,-107.850,174.924,34.592,156.413
C03381=1066.836,376.612,-107.812,174.920,34.586,156.411
C03382=1066.829,376.365,-107.773,174.914,34.579,156.410
C03383=1066.823,376.118,-107.734,174.910,34.573,156.408
C03384=1066.816,375.871,-107.695,174.906,34.566,156.407
C03385=1066.808,375.624,-107.656,174.901,34.559,156.405
C03386=1066.801,375.377,-107.616,174.897,34.552,156.404
C03387=1066.795,375.131,-107.577,174.892,34.546,156.402
C03388=1066.788,374.884,-107.539,174.888,34.539,156.401
C03389=1066.781,374.637,-107.500,174.883,34.533,156.399
C03390=1066.774,374.390,-107.461,174.879,34.526,156.398
C03391=1066.768,374.143,-107.423,174.875,34.520,156.397
C03392=1066.760,373.896,-107.385,174.870,34.514,156.395
C03393=1066.753,373.655,-107.346,174.866,34.507,156.394
C03394=1066.747,373.414,-107.308,174.861,34.501,156.392
C03395=1066.740,373.172,-107.271,174.857,34.494,156.391
C03396=1066.734,372.930,-107.232,174.853,34.488,156.390
C03397=1066.727,372.688,-107.195,174.848,34.481,156.388
C03398=1066.720,372.447,-107.157,174.844,34.475,156.387
C03399=1066.714,372.206,-107.120,174.839,34.469,156.385
C03400=1066.706,371.964,-107.083,174.835,34.463,156.384
C03401=1066.700,371.717,-107.044,174.831,34.457,156.383
C03402=1066.693,371.470,-107.005,174.826,34.450,156.381
C03403=1066.686,371.223,-106.968,174.822,34.444,156.380
C03404=1066.679,370.976,-106.929,174.818,34.438,156.379
C03405=1066.671,370.730,-106.890,174.813,34.432,156.377
C03406=1066.665,370.482,-106.852,174.809,34.425,156.376
C03407=1066.658,370.236,-106.813,174.804,34.419,156.374
C03408=1066.651,369.989,-106.776,174.800,34.412,156.373
C03409=1066.644,369.742,-106.737,174.796,34.406,156.372
C03410=1066.638,369.495,-106.699,174.791,34.400,156.370
C03411=1066.630,369.248,-106.661,174.787,34.394,156.369
C03412=1066.624,369.001,-106.623,174.783,34.387,156.368
C03413=1066.617,368.754,-106.585,174.778,34.381,156.366
C03414=1066.610,368.507,-106.547,174.774,34.375,156.365
C03415=1066.603,368.260,-106.509,174.769,34.369,156.363
C03416=1066.597,368.013,-106.471,174.765,34.363,156.362
C03417=1066.590,367.766,-106.433,174.761,34.357,156.361
C03418=1066.583,367.519,-106.395,174.756,34.351,156.360
C03419=1066.576,367.272,-106.357,174.752,34.344,156.358
C03420=1066.569,367.026,-106.319,174.748,34.338,156.357
C03421=1066.563,366.778,-106.281,174.743,34.332,156.355
C03422=1066.555,366.531,-106.243,174.739,34.326,156.354
C03423=1066.549,366.284,-106.205,174.735,34.320,156.353
C03424=1066.543,366.037,-106.167,174.730,34.314,156.351
C03425=1066.535,365.791,-106.129,174.727,34.307,156.350
C03426=1066.529,365.543,-106.091,174.723,34.302,156.349
C03427=1066.522,365.297,-106.054,174.718,34.295,156.348
C03428=1066.516,365.049,-106.016,174.714,34.289,156.346
C03429=1066.509,364.802,-105.978,174.710,34.283,156.345
C03430=1066.503,364.555,-105.941,174.705,34.277,156.344
C03431=1066.495,364.308,-105.903,174.701,34.271,156.342
C03432=1066.488,364.061,-105.865,174.697,34.265,156.341
C03433=1066.482,363.814,-105.827,174.692,34.259,156.340
C03434=1066.475,363.567,-105.790,174.688,34.253,156.338
C03435=1066.468,363.320,-105.753,174.685,34.248,156.337
C03436=1066.461,363.073,-105.715,174.681,34.241,156.336
C03437=1066.455,362.826,-105.678,174.676,34.236,156.335
C03438=1066.448,362.579,-105.641,174.672,34.230,156.333
C03439=1066.442,362.332,-105.603,174.668,34.224,156.332
C03440=1066.435,362.085,-105.565,174.663,34.218,156.331
C03441=1066.427,361.838,-105.528,174.659,34.212,156.330
C03442=1066.421,361.590,-105.491,174.656,34.206,156.328
C03443=1066.414,361.343,-105.454,174.651,34.200,156.327
C03444=1066.408,361.097,-105.416,174.647,34.194,156.326
C03445=1066.401,360.849,-105.379,174.643,34.189,156.325
C03446=1066.394,360.602,-105.342,174.639,34.183,156.323
C03447=1066.387,360.355,-105.305,174.634,34.177,156.322
C03448=1066.381,360.107,-105.267,174.631,34.171,156.321
C03449=1066.374,359.875,-105.233,174.627,34.166,156.320
C03450=1066.368,359.642,-105.197,174.622,34.160,156.318
C03451=1066.362,359.409,-105.162,174.619,34.155,156.317
C03452=1066.355,359.177,-105.127,174.615,34.149,156.316
C03453=1066.349,358.944,-105.092,174.612,34.144,156.315
C03454=1066.343,358.710,-105.057,174.607,34.138,156.314
C03455=1066.336,358.478,-105.023,174.603,34.133,156.313
C03456=1066.330,358.245,-104.988,174.600,34.128,156.312
C03457=1066.324,357.997,-104.951,174.596,34.122,156.310
C03458=1066.317,357.751,-104.914,174.591,34.116,156.309
C03459=1066.310,357.503,-104.877,174.587,34.111,156.308
C03460=1066.303,357.257,-104.840,174.584,34.105,156.307
C03461=1066.296,357.009,-104.803,174.580,34.099,156.305
C03462=1066.290,356.762,-104.766,174.575,34.094,156.304
C03463=1066.283,356.514,-104.730,174.571,34.088,156.303
C03464=1066.276,356.268,-104.692,174.568,34.083,156.302
C03465=1066.269,356.020,-104.656,174.564,34.077,156.301
C03466=1066.263,355.773,-104.619,174.559,34.071,156.299
C03467=1066.257,355.526,-104.583,174.555,34.066,156.298
C03468=1066.250,355.279,-104.545,174.552,34.060,156.297
C03469=1066.243,355.032,-104.509,174.548,34.054,156.296
C03470=1066.236,354.784,-104.472,174.543,34.049,156.295
C03471=1066.230,354.537,-104.436,174.539,34.043,156.294
C03472=1066.224,354.290,-104.399,174.536,34.038,156.292
C03473=1066.217,354.042,-104.362,174.532,34.032,156.291
C03474=1066.210,353.795,-104.326,174.527,34.027,156.290
C03475=1066.204,353.548,-104.289,174.524,34.021,156.289
C03476=1066.197,353.300,-104.253,174.520,34.016,156.288
C03477=1066.191,353.053,-104.216,174.516,34.010,156.287
C03478=1066.184,352.806,-104.180,174.511,34.004,156.285
C03479=1066.177,352.559,-104.144,174.508,33.999,156.284
C03480=1066.170,352.312,-104.107,174.504,33.993,156.283
C03481=1066.164,352.064,-104.071,174.500,33.988,156.282
C03482=1066.158,351.817,-104.034,174.497,33.982,156.281
C03483=1066.151,351.570,-103.997,174.492,33.977,156.280
C03484=1066.144,351.323,-103.961,174.488,33.972,156.279
C03485=1066.137,351.076,-103.925,174.485,33.966,156.277
C03486=1066.131,350.829,-103.889,174.481,33.961,156.276
C03487=1066.124,350.580,-103.852,174.476,33.956,156.275
C03488=1066.117,350.334,-103.817,174.473,33.950,156.274
C03489=1066.111,350.087,-103.780,174.469,33.945,156.273
C03490=1066.105,349.840,-103.744,174.465,33.939,156.272
C03491=1066.098,349.591,-103.708,174.462,33.934,156.271
C03492=1066.091,349.344,-103.672,174.457,33.928,156.269
C03493=1066.085,349.097,-103.635,174.453,33.923,156.268
C03494=1066.079,348.850,-103.600,174.450,33.918,156.267
C03495=1066.072,348.603,-103.564,174.446,33.912,156.266
C03496=1066.065,348.355,-103.528,174.442,33.907,156.265
C03497=1066.059,348.108,-103.491,174.438,33.902,156.264
C03498=1066.051,347.861,-103.455,174.434,33.896,156.263
C03499=1066.045,347.613,-103.420,174.431,33.891,156.262
C03500=1066.039,347.366,-103.383,174.427,33.886,156.261
C03501=1066.032,347.119,-103.348,174.423,33.880,156.259
C03502=1066.026,346.872,-103.312,174.419,33.875,156.258
C03503=1066.020,346.624,-103.276,174.415,33.870,156.257
C03504=1066.012,346.377,-103.240,174.412,33.865,156.256
C03505=1066.006,346.146,-103.206,174.408,33.860,156.255
C03506=1066.001,345.915,-103.173,174.405,33.855,156.254
C03507=1065.995,345.684,-103.140,174.400,33.850,156.253
C03508=1065.989,345.453,-103.107,174.397,33.845,156.252
C03509=1065.983,345.222,-103.073,174.394,33.840,156.251
C03510=1065.976,344.991,-103.039,174.390,33.835,156.250
C03511=1065.970,344.761,-103.006,174.387,33.830,156.249
C03512=1065.964,344.530,-102.973,174.384,33.826,156.248
C03513=1065.958,344.282,-102.937,174.379,33.820,156.247
C03514=1065.951,344.035,-102.902,174.376,33.815,156.246
C03515=1065.945,343.787,-102.866,174.372,33.810,156.245
C03516=1065.938,343.541,-102.831,174.369,33.805,156.244
C03517=1065.932,343.293,-102.795,174.365,33.799,156.243
C03518=1065.925,343.046,-102.760,174.361,33.795,156.242
C03519=1065.919,342.798,-102.725,174.357,33.789,156.241
C03520=1065.913,342.550,-102.689,174.353,33.784,156.239
C03521=1065.906,342.303,-102.654,174.350,33.779,156.238
C03522=1065.900,342.055,-102.618,174.346,33.774,156.237
C03523=1065.893,341.808,-102.583,174.343,33.769,156.236
C03524=1065.886,341.561,-102.547,174.339,33.764,156.235
C03525=1065.880,341.314,-102.511,174.335,33.759,156.234
C03526=1065.873,341.066,-102.476,174.331,33.754,156.233
C03527=1065.866,340.819,-102.441,174.328,33.749,156.232
C03528=1065.860,340.571,-102.405,174.324,33.743,156.231
C03529=1065.854,340.324,-102.370,174.321,33.739,156.230
C03530=1065.847,340.076,-102.336,174.317,33.733,156.229
C03531=1065.840,339.829,-102.301,174.313,33.728,156.228
C03532=1065.834,339.581,-102.265,174.309,33.723,156.227
C03533=1065.827,339.334,-102.230,174.306,33.718,156.226
C03534=1065.821,339.086,-102.195,174.302,33.713,156.225
C03535=1065.815,338.839,-102.159,174.299,33.708,156.224
C03536=1065.809,338.592,-102.124,174.295,33.703,156.223
C03537=1065.802,338.344,-102.089,174.292,33.698,156.222
C03538=1065.796,338.096,-102.054,174.287,33.693,156.221
C03539=1065.789,337.849,-102.019,174.284,33.688,156.220
C03540=1065.782,337.601,-101.984,174.280,33.683,156.219
C03541=1065.776,337.355,-101.949,174.277,33.678,156.218
C03542=1065.770,337.107,-101.914,174.273,33.673,156.217
C03543=1065.764,336.859,-101.879,174.270,33.668,156.216
C03544=1065.757,336.612,-101.844,174.266,33.663,156.215
C03545=1065.751,336.364,-101.809,174.262,33.658,156.214
C03546=1065.744,336.116,-101.774,174.258,33.653,156.213
C03547=1065.738,335.870,-101.739,174.255,33.648,156.212
C03548=1065.731,335.622,-101.705,174.252,33.644,156.211
C03549=1065.724,335.374,-101.670,174.248,33.639,156.210
C03550=1065.718,335.126,-101.635,174.245,33.634,156.209
C03551=1065.711,334.879,-101.600,174.241,33.629,156.208
C03552=1065.705,334.632,-101.566,174.238,33.624,156.207
C03553=1065.699,334.384,-101.531,174.233,33.619,156.206
C03554=1065.692,334.136,-101.497,174.230,33.614,156.205
C03555=1065.685,333.889,-101.461,174.227,33.609,156.204
C03556=1065.679,333.642,-101.427,174.223,33.604,156.203
C03557=1065.673,333.394,-101.392,174.220,33.600,156.202
C03558=1065.666,333.146,-101.358,174.216,33.595,156.201
C03559=1065.660,332.899,-101.324,174.213,33.590,156.200
C03560=1065.654,332.652,-101.289,174.210,33.585,156.199
C03561=1065.648,332.418,-101.255,174.205,33.580,156.198
C03562=1065.642,332.185,-101.223,174.202,33.576,156.197
C03563=1065.636,331.951,-101.191,174.199,33.571,156.196
C03564=1065.630,331.719,-101.158,174.196,33.567,156.195
C03565=1065.624,331.485,-101.126,174.193,33.562,156.194
C03566=1065.618,331.251,-101.093,174.189,33.558,156.193
C03567=1065.612,331.018,-101.060,174.186,33.553,156.192
C03568=1065.606,330.784,-101.029,174.183,33.548,156.191
C03569=1065.600,330.538,-100.994,174.180,33.544,156.190
C03570=1065.593,330.290,-100.960,174.175,33.539,156.189
C03571=1065.586,330.042,-100.926,174.172,33.534,156.188
C03572=1065.580,329.794,-100.891,174.169,33.530,156.188
C03573=1065.573,329.547,-100.858,174.165,33.525,156.187
C03574=1065.567,329.299,-100.823,174.162,33.521,156.186
C03575=1065.560,329.051,-100.789,174.158,33.516,156.185
C03576=1065.553,328.804,-100.755,174.155,33.511,156.184
C03577=1065.547,328.556,-100.721,174.152,33.507,156.183
C03578=1065.541,328.309,-100.687,174.148,33.502,156.182
C03579=1065.534,328.062,-100.652,174.145,33.497,156.181
C03580=1065.528,327.813,-100.619,174.141,33.492,156.180
C03581=1065.521,327.566,-100.585,174.137,33.488,156.179
C03582=1065.514,327.318,-100.551,174.134,33.483,156.178
C03583=1065.509,327.071,-100.517,174.131,33.479,156.177
C03584=1065.501,326.823,-100.483,174.127,33.474,156.176
C03585=1065.495,326.575,-100.448,174.124,33.469,156.175
C03586=1065.488,326.328,-100.415,174.121,33.464,156.174
C03587=1065.482,326.080,-100.381,174.117,33.460,156.174
C03588=1065.476,325.833,-100.347,174.114,33.455,156.173
C03589=1065.469,325.585,-100.313,174.111,33.451,156.172
C03590=1065.463,325.338,-100.279,174.107,33.446,156.171
C03591=1065.456,325.090,-100.246,174.103,33.441,156.170
C03592=1065.450,324.843,-100.211,174.100,33.437,156.169
C03593=1065.444,324.595,-100.177,174.096,33.432,156.168
C03594=1065.437,324.348,-100.144,174.093,33.428,156.167
C03595=1065.431,324.099,-100.110,174.090,33.423,156.166
C03596=1065.424,323.852,-100.076,174.087,33.418,156.165
C03597=1065.418,323.604,-100.042,174.083,33.413,156.164
C03598=1065.411,323.357,-100.009,174.080,33.409,156.163
C03599=1065.406,323.109,-99.975,174.077,33.405,156.163
C03600=1065.399,322.862,-99.941,174.074,33.400,156.162
C03601=1065.393,322.614,-99.907,174.070,33.395,156.161
C03602=1065.387,322.366,-99.874,174.067,33.391,156.160
C03603=1065.380,322.119,-99.840,174.063,33.386,156.159
C03604=1065.374,321.871,-99.807,174.060,33.381,156.158
C03605=1065.367,321.623,-99.773,174.056,33.377,156.157
C03606=1065.362,321.375,-99.740,174.053,33.372,156.156
C03607=1065.354,321.128,-99.706,174.050,33.368,156.155
C03608=1065.349,320.880,-99.672,174.047,33.363,156.154
C03609=1065.342,320.633,-99.639,174.043,33.359,156.153
C03610=1065.336,320.385,-99.605,174.040,33.354,156.152
C03611=1065.330,320.137,-99.572,174.037,33.349,156.152
C03612=1065.324,319.890,-99.538,174.034,33.345,156.151
C03613=1065.317,319.642,-99.505,174.030,33.340,156.150
C03614=1065.311,319.394,-99.471,174.027,33.336,156.149
C03615=1065.305,319.147,-99.438,174.024,33.331,156.148
C03616=1065.299,318.899,-99.405,174.021,33.327,156.147
C03617=1065.292,318.662,-99.372,174.017,33.323,156.146
C03618=1065.287,318.426,-99.341,174.014,33.318,156.145
